LIN {X 151.987,Y 68.741,Z 52.000,A 180.000,B 0.000,C 180.000} C_DIS
LIN {X 152.500,Y 68.741,Z 52.000,A 180.000,B 0.000,C 180.000} C_DIS
LIN {X 152.500,Y 68.741,Z 45.000,A 180.000,B 0.000,C 180.000} C_DIS
LIN {X 155.010,Y 68.741,Z 45.000,A 180.000,B 0.000,C 180.000} C_DIS
; Link Move Starts
LIN {X 155.120,Y 68.741,Z 45.026,A 180.000,B 0.000,C 180.000} C_DIS
LIN {X 155.230,Y 68.741,Z 45.051,A 180.000,B 0.000,C 180.000} C_DIS
LIN {X 155.771,Y 69.054,Z 45.051,A 180.000,B 0.000,C 180.000} C_DIS
LIN {X 155.771,Y 69.679,Z 45.051,A 180.000,B 0.000,C 180.000} C_DIS
LIN {X 155.230,Y 69.991,Z 45.051,A 180.000,B 0.000,C 180.000} C_DIS
LIN {X 155.120,Y 69.991,Z 45.026,A 180.000,B 0.000,C 180.000} C_DIS
LIN {X 155.010,Y 69.991,Z 45.000,A 180.000,B 0.000,C 180.000} C_DIS
; Cutting Move Starts
LIN {X 152.500,Y 69.991,Z 45.000,A 180.000,B 0.000,C 180.000} C_DIS
LIN {X 152.500,Y 69.991,Z 52.000,A 180.000,B 0.000,C 180.000} C_DIS
LIN {X 152.119,Y 69.991,Z 52.000,A 180.000,B 0.000,C 180.000} C_DIS
LIN {X 152.117,Y 69.991,Z 57.000,A 180.000,B 0.000,C 180.000} C_DIS
LIN {X 138.527,Y 69.991,Z 57.000,A 180.000,B 0.000,C 180.000} C_DIS
LIN {X 138.527,Y 69.991,Z 62.000,A 180.000,B 0.000,C 180.000} C_DIS
LIN {X 64.935,Y 69.991,Z 62.000,A 180.000,B 0.000,C 180.000} C_DIS
LIN {X 64.931,Y 69.991,Z 82.040,A 180.000,B 0.000,C 180.000} C_DIS
LIN {X 64.891,Y 69.991,Z 82.144,A 180.000,B 0.000,C 180.000} C_DIS
LIN {X 64.812,Y 69.991,Z 82.250,A 180.000,B 0.000,C 180.000} C_DIS
LIN {X 64.651,Y 69.991,Z 82.406,A 180.000,B 0.000,C 180.000} C_DIS
LIN {X 64.413,Y 69.991,Z 82.569,A 180.000,B 0.000,C 180.000} C_DIS
LIN {X 64.256,Y 69.991,Z 82.658,A 180.000,B 0.000,C 180.000} C_DIS
LIN {X 63.886,Y 69.991,Z 82.826,A 180.000,B 0.000,C 180.000} C_DIS
LIN {X 63.427,Y 69.991,Z 82.974,A 180.000,B 0.000,C 180.000} C_DIS
LIN {X 63.116,Y 69.991,Z 83.044,A 180.000,B 0.000,C 180.000} C_DIS
LIN {X 62.751,Y 69.991,Z 83.103,A 180.000,B 0.000,C 180.000} C_DIS
LIN {X 62.375,Y 69.991,Z 83.137,A 180.000,B 0.000,C 180.000} C_DIS
LIN {X 62.046,Y 69.991,Z 83.148,A 180.000,B 0.000,C 180.000} C_DIS
LIN {X 57.054,Y 69.991,Z 83.146,A 180.000,B 0.000,C 180.000} C_DIS
LIN {X 56.742,Y 69.991,Z 83.135,A 180.000,B 0.000,C 180.000} C_DIS
LIN {X 56.417,Y 69.991,Z 83.115,A 180.000,B 0.000,C 180.000} C_DIS
LIN {X 56.096,Y 69.991,Z 83.085,A 180.000,B 0.000,C 180.000} C_DIS
LIN {X 55.739,Y 69.991,Z 83.040,A 180.000,B 0.000,C 180.000} C_DIS
LIN {X 55.361,Y 69.991,Z 82.981,A 180.000,B 0.000,C 180.000} C_DIS
LIN {X 55.002,Y 69.991,Z 82.912,A 180.000,B 0.000,C 180.000} C_DIS
LIN {X 54.625,Y 69.991,Z 82.827,A 180.000,B 0.000,C 180.000} C_DIS
LIN {X 54.239,Y 69.991,Z 82.728,A 180.000,B 0.000,C 180.000} C_DIS
LIN {X 53.862,Y 69.991,Z 82.617,A 180.000,B 0.000,C 180.000} C_DIS
LIN {X 53.473,Y 69.991,Z 82.491,A 180.000,B 0.000,C 180.000} C_DIS
LIN {X 53.083,Y 69.991,Z 82.351,A 180.000,B 0.000,C 180.000} C_DIS
LIN {X 52.690,Y 69.991,Z 82.196,A 180.000,B 0.000,C 180.000} C_DIS
LIN {X 52.293,Y 69.991,Z 82.027,A 180.000,B 0.000,C 180.000} C_DIS
LIN {X 51.893,Y 69.991,Z 81.843,A 180.000,B 0.000,C 180.000} C_DIS
LIN {X 51.488,Y 69.991,Z 81.643,A 180.000,B 0.000,C 180.000} C_DIS
LIN {X 51.080,Y 69.991,Z 81.428,A 180.000,B 0.000,C 180.000} C_DIS
LIN {X 50.671,Y 69.991,Z 81.199,A 180.000,B 0.000,C 180.000} C_DIS
LIN {X 50.251,Y 69.991,Z 80.950,A 180.000,B 0.000,C 180.000} C_DIS
LIN {X 49.826,Y 69.991,Z 80.683,A 180.000,B 0.000,C 180.000} C_DIS
LIN {X 49.494,Y 69.991,Z 80.467,A 180.000,B 0.000,C 180.000} C_DIS
LIN {X 49.494,Y 69.991,Z 62.000,A 180.000,B 0.000,C 180.000} C_DIS
LIN {X 16.473,Y 69.991,Z 62.000,A 180.000,B 0.000,C 180.000} C_DIS
LIN {X 16.473,Y 69.991,Z 57.000,A 180.000,B 0.000,C 180.000} C_DIS
LIN {X 2.881,Y 69.991,Z 57.000,A 180.000,B 0.000,C 180.000} C_DIS
LIN {X 2.881,Y 69.991,Z 52.000,A 180.000,B 0.000,C 180.000} C_DIS
LIN {X 2.500,Y 69.991,Z 52.000,A 180.000,B 0.000,C 180.000} C_DIS
LIN {X 2.500,Y 69.991,Z 45.000,A 180.000,B 0.000,C 180.000} C_DIS
LIN {X -0.010,Y 69.991,Z 45.000,A 180.000,B 0.000,C 180.000} C_DIS
; Link Move Starts
LIN {X -0.120,Y 69.991,Z 45.026,A 180.000,B 0.000,C 180.000} C_DIS
LIN {X -0.230,Y 69.991,Z 45.051,A 180.000,B 0.000,C 180.000} C_DIS
LIN {X -0.771,Y 70.304,Z 45.051,A 180.000,B 0.000,C 180.000} C_DIS
LIN {X -0.771,Y 70.929,Z 45.051,A 180.000,B 0.000,C 180.000} C_DIS
LIN {X -0.230,Y 71.241,Z 45.051,A 180.000,B 0.000,C 180.000} C_DIS
LIN {X -0.120,Y 71.241,Z 45.026,A 180.000,B 0.000,C 180.000} C_DIS
LIN {X -0.010,Y 71.241,Z 45.000,A 180.000,B 0.000,C 180.000} C_DIS
; Cutting Move Starts
LIN {X 2.500,Y 71.241,Z 45.000,A 180.000,B 0.000,C 180.000} C_DIS
LIN {X 2.500,Y 71.241,Z 52.000,A 180.000,B 0.000,C 180.000} C_DIS
LIN {X 2.765,Y 71.241,Z 52.000,A 180.000,B 0.000,C 180.000} C_DIS
LIN {X 2.767,Y 71.241,Z 57.000,A 180.000,B 0.000,C 180.000} C_DIS
LIN {X 15.220,Y 71.241,Z 57.000,A 180.000,B 0.000,C 180.000} C_DIS
LIN {X 15.224,Y 71.241,Z 62.000,A 180.000,B 0.000,C 180.000} C_DIS
LIN {X 49.913,Y 71.241,Z 62.000,A 180.000,B 0.000,C 180.000} C_DIS
LIN {X 49.916,Y 71.241,Z 80.467,A 180.000,B 0.000,C 180.000} C_DIS
LIN {X 50.252,Y 71.241,Z 80.686,A 180.000,B 0.000,C 180.000} C_DIS
LIN {X 50.672,Y 71.241,Z 80.949,A 180.000,B 0.000,C 180.000} C_DIS
LIN {X 51.086,Y 71.241,Z 81.195,A 180.000,B 0.000,C 180.000} C_DIS
LIN {X 51.500,Y 71.241,Z 81.427,A 180.000,B 0.000,C 180.000} C_DIS
LIN {X 51.909,Y 71.241,Z 81.643,A 180.000,B 0.000,C 180.000} C_DIS
LIN {X 52.314,Y 71.241,Z 81.842,A 180.000,B 0.000,C 180.000} C_DIS
LIN {X 52.714,Y 71.241,Z 82.026,A 180.000,B 0.000,C 180.000} C_DIS
LIN {X 53.057,Y 71.241,Z 82.173,A 180.000,B 0.000,C 180.000} C_DIS
LIN {X 53.316,Y 71.241,Z 82.278,A 180.000,B 0.000,C 180.000} C_DIS
LIN {X 53.758,Y 71.241,Z 82.442,A 180.000,B 0.000,C 180.000} C_DIS
LIN {X 54.177,Y 71.241,Z 82.579,A 180.000,B 0.000,C 180.000} C_DIS
LIN {X 54.617,Y 71.241,Z 82.706,A 180.000,B 0.000,C 180.000} C_DIS
LIN {X 55.075,Y 71.241,Z 82.819,A 180.000,B 0.000,C 180.000} C_DIS
LIN {X 55.690,Y 71.241,Z 82.942,A 180.000,B 0.000,C 180.000} C_DIS
LIN {X 56.199,Y 71.241,Z 83.020,A 180.000,B 0.000,C 180.000} C_DIS
LIN {X 56.683,Y 71.241,Z 83.076,A 180.000,B 0.000,C 180.000} C_DIS
LIN {X 57.277,Y 71.241,Z 83.123,A 180.000,B 0.000,C 180.000} C_DIS
LIN {X 57.978,Y 71.241,Z 83.146,A 180.000,B 0.000,C 180.000} C_DIS
LIN {X 61.059,Y 71.241,Z 83.147,A 180.000,B 0.000,C 180.000} C_DIS
LIN {X 61.178,Y 71.241,Z 83.135,A 180.000,B 0.000,C 180.000} C_DIS
LIN {X 61.226,Y 71.241,Z 83.119,A 180.000,B 0.000,C 180.000} C_DIS
LIN {X 61.230,Y 71.241,Z 62.000,A 180.000,B 0.000,C 180.000} C_DIS
LIN {X 73.375,Y 71.241,Z 62.000,A 180.000,B 0.000,C 180.000} C_DIS
LIN {X 73.375,Y 71.241,Z 57.000,A 180.000,B 0.000,C 180.000} C_DIS
LIN {X 81.625,Y 71.241,Z 57.000,A 180.000,B 0.000,C 180.000} C_DIS
LIN {X 81.625,Y 71.241,Z 62.000,A 180.000,B 0.000,C 180.000} C_DIS
LIN {X 139.775,Y 71.241,Z 62.000,A 180.000,B 0.000,C 180.000} C_DIS
LIN {X 139.777,Y 71.241,Z 57.000,A 180.000,B 0.000,C 180.000} C_DIS
LIN {X 152.233,Y 71.241,Z 57.000,A 180.000,B 0.000,C 180.000} C_DIS
LIN {X 152.233,Y 71.241,Z 52.000,A 180.000,B 0.000,C 180.000} C_DIS
LIN {X 152.500,Y 71.241,Z 52.000,A 180.000,B 0.000,C 180.000} C_DIS
LIN {X 152.500,Y 71.241,Z 45.000,A 180.000,B 0.000,C 180.000} C_DIS
LIN {X 155.010,Y 71.241,Z 45.000,A 180.000,B 0.000,C 180.000} C_DIS
; Link Move Starts
LIN {X 155.120,Y 71.241,Z 45.026,A 180.000,B 0.000,C 180.000} C_DIS
LIN {X 155.230,Y 71.241,Z 45.051,A 180.000,B 0.000,C 180.000} C_DIS
LIN {X 155.771,Y 71.553,Z 45.051,A 180.000,B 0.000,C 180.000} C_DIS
LIN {X 155.771,Y 72.178,Z 45.051,A 180.000,B 0.000,C 180.000} C_DIS
LIN {X 155.230,Y 72.491,Z 45.051,A 180.000,B 0.000,C 180.000} C_DIS
LIN {X 155.120,Y 72.491,Z 45.026,A 180.000,B 0.000,C 180.000} C_DIS
LIN {X 155.010,Y 72.491,Z 45.000,A 180.000,B 0.000,C 180.000} C_DIS
; Cutting Move Starts
LIN {X 152.500,Y 72.491,Z 45.000,A 180.000,B 0.000,C 180.000} C_DIS
LIN {X 152.500,Y 72.491,Z 52.000,A 180.000,B 0.000,C 180.000} C_DIS
LIN {X 152.330,Y 72.491,Z 52.000,A 180.000,B 0.000,C 180.000} C_DIS
LIN {X 152.330,Y 72.491,Z 57.000,A 180.000,B 0.000,C 180.000} C_DIS
LIN {X 141.026,Y 72.491,Z 57.000,A 180.000,B 0.000,C 180.000} C_DIS
LIN {X 141.026,Y 72.491,Z 62.000,A 180.000,B 0.000,C 180.000} C_DIS
LIN {X 83.076,Y 72.491,Z 62.000,A 180.000,B 0.000,C 180.000} C_DIS
LIN {X 83.076,Y 72.491,Z 57.000,A 180.000,B 0.000,C 180.000} C_DIS
LIN {X 71.924,Y 72.491,Z 57.000,A 180.000,B 0.000,C 180.000} C_DIS
LIN {X 71.924,Y 72.491,Z 62.000,A 180.000,B 0.000,C 180.000} C_DIS
LIN {X 57.525,Y 72.491,Z 62.000,A 180.000,B 0.000,C 180.000} C_DIS
LIN {X 57.521,Y 72.491,Z 82.696,A 180.000,B 0.000,C 180.000} C_DIS
LIN {X 57.489,Y 72.491,Z 82.734,A 180.000,B 0.000,C 180.000} C_DIS
LIN {X 57.421,Y 72.491,Z 82.763,A 180.000,B 0.000,C 180.000} C_DIS
LIN {X 57.262,Y 72.491,Z 82.785,A 180.000,B 0.000,C 180.000} C_DIS
LIN {X 56.970,Y 72.491,Z 82.787,A 180.000,B 0.000,C 180.000} C_DIS
LIN {X 56.506,Y 72.491,Z 82.752,A 180.000,B 0.000,C 180.000} C_DIS
LIN {X 55.884,Y 72.491,Z 82.665,A 180.000,B 0.000,C 180.000} C_DIS
LIN {X 55.297,Y 72.491,Z 82.553,A 180.000,B 0.000,C 180.000} C_DIS
LIN {X 54.770,Y 72.491,Z 82.429,A 180.000,B 0.000,C 180.000} C_DIS
LIN {X 54.285,Y 72.491,Z 82.296,A 180.000,B 0.000,C 180.000} C_DIS
LIN {X 53.823,Y 72.491,Z 82.152,A 180.000,B 0.000,C 180.000} C_DIS
LIN {X 53.356,Y 72.491,Z 81.988,A 180.000,B 0.000,C 180.000} C_DIS
LIN {X 52.884,Y 72.491,Z 81.804,A 180.000,B 0.000,C 180.000} C_DIS
LIN {X 52.420,Y 72.491,Z 81.604,A 180.000,B 0.000,C 180.000} C_DIS
LIN {X 51.957,Y 72.491,Z 81.385,A 180.000,B 0.000,C 180.000} C_DIS
LIN {X 51.493,Y 72.491,Z 81.145,A 180.000,B 0.000,C 180.000} C_DIS
LIN {X 51.033,Y 72.491,Z 80.888,A 180.000,B 0.000,C 180.000} C_DIS
LIN {X 50.578,Y 72.491,Z 80.613,A 180.000,B 0.000,C 180.000} C_DIS
LIN {X 50.346,Y 72.491,Z 80.467,A 180.000,B 0.000,C 180.000} C_DIS
LIN {X 50.346,Y 72.491,Z 62.000,A 180.000,B 0.000,C 180.000} C_DIS
LIN {X 13.974,Y 72.491,Z 62.000,A 180.000,B 0.000,C 180.000} C_DIS
LIN {X 13.974,Y 72.491,Z 57.000,A 180.000,B 0.000,C 180.000} C_DIS
LIN {X 2.670,Y 72.491,Z 57.000,A 180.000,B 0.000,C 180.000} C_DIS
LIN {X 2.670,Y 72.491,Z 52.000,A 180.000,B 0.000,C 180.000} C_DIS
LIN {X 2.500,Y 72.491,Z 52.000,A 180.000,B 0.000,C 180.000} C_DIS
LIN {X 2.495,Y 72.491,Z 45.000,A 180.000,B 0.000,C 180.000} C_DIS
LIN {X -0.010,Y 72.491,Z 45.000,A 180.000,B 0.000,C 180.000} C_DIS
; Link Move Starts
LIN {X -0.120,Y 72.491,Z 45.026,A 180.000,B 0.000,C 180.000} C_DIS
LIN {X -0.230,Y 72.491,Z 45.051,A 180.000,B 0.000,C 180.000} C_DIS
LIN {X -0.771,Y 72.803,Z 45.051,A 180.000,B 0.000,C 180.000} C_DIS
LIN {X -0.771,Y 73.428,Z 45.051,A 180.000,B 0.000,C 180.000} C_DIS
LIN {X -0.230,Y 73.741,Z 45.051,A 180.000,B 0.000,C 180.000} C_DIS
LIN {X -0.120,Y 73.741,Z 45.026,A 180.000,B 0.000,C 180.000} C_DIS
LIN {X -0.010,Y 73.741,Z 45.000,A 180.000,B 0.000,C 180.000} C_DIS
; Cutting Move Starts
LIN {X 2.500,Y 73.741,Z 45.000,A 180.000,B 0.000,C 180.000} C_DIS
LIN {X 2.500,Y 73.741,Z 52.000,A 180.000,B 0.000,C 180.000} C_DIS
LIN {X 2.597,Y 73.741,Z 52.000,A 180.000,B 0.000,C 180.000} C_DIS
LIN {X 2.597,Y 73.741,Z 57.000,A 180.000,B 0.000,C 180.000} C_DIS
LIN {X 12.724,Y 73.741,Z 57.000,A 180.000,B 0.000,C 180.000} C_DIS
LIN {X 12.724,Y 73.741,Z 62.000,A 180.000,B 0.000,C 180.000} C_DIS
LIN {X 51.532,Y 73.741,Z 62.000,A 180.000,B 0.000,C 180.000} C_DIS
LIN {X 51.533,Y 73.741,Z 80.467,A 180.000,B 0.000,C 180.000} C_DIS
LIN {X 51.861,Y 73.741,Z 80.604,A 180.000,B 0.000,C 180.000} C_DIS
LIN {X 52.317,Y 73.741,Z 80.775,A 180.000,B 0.000,C 180.000} C_DIS
LIN {X 52.750,Y 73.741,Z 80.905,A 180.000,B 0.000,C 180.000} C_DIS
LIN {X 53.082,Y 73.741,Z 80.979,A 180.000,B 0.000,C 180.000} C_DIS
LIN {X 53.328,Y 73.741,Z 81.008,A 180.000,B 0.000,C 180.000} C_DIS
LIN {X 53.527,Y 73.741,Z 81.004,A 180.000,B 0.000,C 180.000} C_DIS
LIN {X 53.649,Y 73.741,Z 80.977,A 180.000,B 0.000,C 180.000} C_DIS
LIN {X 53.735,Y 73.741,Z 80.931,A 180.000,B 0.000,C 180.000} C_DIS
LIN {X 53.786,Y 73.741,Z 80.873,A 180.000,B 0.000,C 180.000} C_DIS
LIN {X 53.816,Y 73.741,Z 80.795,A 180.000,B 0.000,C 180.000} C_DIS
LIN {X 53.820,Y 73.741,Z 62.000,A 180.000,B 0.000,C 180.000} C_DIS
LIN {X 71.016,Y 73.741,Z 62.000,A 180.000,B 0.000,C 180.000} C_DIS
LIN {X 71.016,Y 73.741,Z 57.000,A 180.000,B 0.000,C 180.000} C_DIS
LIN {X 83.984,Y 73.741,Z 57.000,A 180.000,B 0.000,C 180.000} C_DIS
LIN {X 83.984,Y 73.741,Z 62.000,A 180.000,B 0.000,C 180.000} C_DIS
LIN {X 142.272,Y 73.741,Z 62.000,A 180.000,B 0.000,C 180.000} C_DIS
LIN {X 142.276,Y 73.741,Z 57.000,A 180.000,B 0.000,C 180.000} C_DIS
LIN {X 152.403,Y 73.741,Z 57.000,A 180.000,B 0.000,C 180.000} C_DIS
LIN {X 152.403,Y 73.741,Z 52.000,A 180.000,B 0.000,C 180.000} C_DIS
LIN {X 152.500,Y 73.741,Z 52.000,A 180.000,B 0.000,C 180.000} C_DIS
LIN {X 152.500,Y 73.741,Z 45.000,A 180.000,B 0.000,C 180.000} C_DIS
LIN {X 155.010,Y 73.741,Z 45.000,A 180.000,B 0.000,C 180.000} C_DIS
; Link Move Starts
LIN {X 155.120,Y 73.741,Z 45.026,A 180.000,B 0.000,C 180.000} C_DIS
LIN {X 155.230,Y 73.741,Z 45.051,A 180.000,B 0.000,C 180.000} C_DIS
LIN {X 155.771,Y 74.053,Z 45.051,A 180.000,B 0.000,C 180.000} C_DIS
LIN {X 155.771,Y 74.678,Z 45.051,A 180.000,B 0.000,C 180.000} C_DIS
LIN {X 155.230,Y 74.991,Z 45.051,A 180.000,B 0.000,C 180.000} C_DIS
LIN {X 155.120,Y 74.991,Z 45.026,A 180.000,B 0.000,C 180.000} C_DIS
LIN {X 155.010,Y 74.991,Z 45.000,A 180.000,B 0.000,C 180.000} C_DIS
; Cutting Move Starts
LIN {X 152.500,Y 74.991,Z 45.000,A 180.000,B 0.000,C 180.000} C_DIS
LIN {X 152.500,Y 74.991,Z 52.000,A 180.000,B 0.000,C 180.000} C_DIS
LIN {X 152.453,Y 74.991,Z 52.000,A 180.000,B 0.000,C 180.000} C_DIS
LIN {X 152.453,Y 74.991,Z 57.000,A 180.000,B 0.000,C 180.000} C_DIS
LIN {X 143.526,Y 74.991,Z 57.000,A 180.000,B 0.000,C 180.000} C_DIS
LIN {X 143.526,Y 74.991,Z 62.000,A 180.000,B 0.000,C 180.000} C_DIS
LIN {X 84.563,Y 74.991,Z 62.000,A 180.000,B 0.000,C 180.000} C_DIS
LIN {X 84.563,Y 74.991,Z 57.000,A 180.000,B 0.000,C 180.000} C_DIS
LIN {X 70.437,Y 74.991,Z 57.000,A 180.000,B 0.000,C 180.000} C_DIS
LIN {X 70.436,Y 74.991,Z 62.000,A 180.000,B 0.000,C 180.000} C_DIS
LIN {X 11.474,Y 74.991,Z 62.000,A 180.000,B 0.000,C 180.000} C_DIS
LIN {X 11.474,Y 74.991,Z 57.000,A 180.000,B 0.000,C 180.000} C_DIS
LIN {X 2.547,Y 74.991,Z 57.000,A 180.000,B 0.000,C 180.000} C_DIS
LIN {X 2.547,Y 74.991,Z 52.000,A 180.000,B 0.000,C 180.000} C_DIS
LIN {X 2.500,Y 74.991,Z 52.000,A 180.000,B 0.000,C 180.000} C_DIS
LIN {X 2.500,Y 74.991,Z 45.000,A 180.000,B 0.000,C 180.000} C_DIS
LIN {X -0.010,Y 74.991,Z 45.000,A 180.000,B 0.000,C 180.000} C_DIS
; Link Move Starts
LIN {X -0.120,Y 74.991,Z 45.026,A 180.000,B 0.000,C 180.000} C_DIS
LIN {X -0.230,Y 74.991,Z 45.051,A 180.000,B 0.000,C 180.000} C_DIS
LIN {X -0.771,Y 75.303,Z 45.051,A 180.000,B 0.000,C 180.000} C_DIS
LIN {X -0.771,Y 75.928,Z 45.051,A 180.000,B 0.000,C 180.000} C_DIS
LIN {X -0.230,Y 76.241,Z 45.051,A 180.000,B 0.000,C 180.000} C_DIS
LIN {X -0.120,Y 76.241,Z 45.026,A 180.000,B 0.000,C 180.000} C_DIS
LIN {X -0.010,Y 76.241,Z 45.000,A 180.000,B 0.000,C 180.000} C_DIS
; Cutting Move Starts
LIN {X 2.500,Y 76.241,Z 45.000,A 180.000,B 0.000,C 180.000} C_DIS
LIN {X 2.500,Y 76.241,Z 52.000,A 180.000,B 0.000,C 180.000} C_DIS
LIN {X 2.515,Y 76.241,Z 52.000,A 180.000,B 0.000,C 180.000} C_DIS
LIN {X 2.515,Y 76.241,Z 57.000,A 180.000,B 0.000,C 180.000} C_DIS
LIN {X 10.340,Y 76.241,Z 57.000,A 180.000,B 0.000,C 180.000} C_DIS
LIN {X 10.340,Y 76.241,Z 62.000,A 180.000,B 0.000,C 180.000} C_DIS
LIN {X 70.111,Y 76.241,Z 62.000,A 180.000,B 0.000,C 180.000} C_DIS
LIN {X 70.111,Y 76.241,Z 57.000,A 180.000,B 0.000,C 180.000} C_DIS
LIN {X 84.889,Y 76.241,Z 57.000,A 180.000,B 0.000,C 180.000} C_DIS
LIN {X 84.889,Y 76.241,Z 62.000,A 180.000,B 0.000,C 180.000} C_DIS
LIN {X 144.660,Y 76.241,Z 62.000,A 180.000,B 0.000,C 180.000} C_DIS
LIN {X 144.660,Y 76.241,Z 57.000,A 180.000,B 0.000,C 180.000} C_DIS
LIN {X 152.484,Y 76.241,Z 57.000,A 180.000,B 0.000,C 180.000} C_DIS
LIN {X 152.485,Y 76.241,Z 52.000,A 180.000,B 0.000,C 180.000} C_DIS
LIN {X 152.500,Y 76.241,Z 52.000,A 180.000,B 0.000,C 180.000} C_DIS
LIN {X 152.500,Y 76.241,Z 45.000,A 180.000,B 0.000,C 180.000} C_DIS
LIN {X 155.010,Y 76.241,Z 45.000,A 180.000,B 0.000,C 180.000} C_DIS
; Link Move Starts
LIN {X 155.120,Y 76.241,Z 45.026,A 180.000,B 0.000,C 180.000} C_DIS
LIN {X 155.230,Y 76.241,Z 45.051,A 180.000,B 0.000,C 180.000} C_DIS
LIN {X 155.771,Y 76.553,Z 45.051,A 180.000,B 0.000,C 180.000} C_DIS
LIN {X 155.771,Y 77.178,Z 45.051,A 180.000,B 0.000,C 180.000} C_DIS
LIN {X 155.230,Y 77.490,Z 45.051,A 180.000,B 0.000,C 180.000} C_DIS
LIN {X 155.120,Y 77.490,Z 45.026,A 180.000,B 0.000,C 180.000} C_DIS
LIN {X 155.010,Y 77.490,Z 45.000,A 180.000,B 0.000,C 180.000} C_DIS
; Cutting Move Starts
LIN {X 152.500,Y 77.490,Z 45.000,A 180.000,B 0.000,C 180.000} C_DIS
LIN {X 152.500,Y 77.490,Z 57.000,A 180.000,B 0.000,C 180.000} C_DIS
LIN {X 145.000,Y 77.490,Z 57.000,A 180.000,B 0.000,C 180.000} C_DIS
LIN {X 145.000,Y 77.490,Z 62.000,A 180.000,B 0.000,C 180.000} C_DIS
LIN {X 84.998,Y 77.490,Z 62.000,A 180.000,B 0.000,C 180.000} C_DIS
LIN {X 84.998,Y 77.490,Z 57.000,A 180.000,B 0.000,C 180.000} C_DIS
LIN {X 70.002,Y 77.490,Z 57.000,A 180.000,B 0.000,C 180.000} C_DIS
LIN {X 70.000,Y 77.490,Z 62.000,A 180.000,B 0.000,C 180.000} C_DIS
LIN {X 10.000,Y 77.490,Z 62.000,A 180.000,B 0.000,C 180.000} C_DIS
LIN {X 10.000,Y 77.490,Z 57.000,A 180.000,B 0.000,C 180.000} C_DIS
LIN {X 2.500,Y 77.490,Z 57.000,A 180.000,B 0.000,C 180.000} C_DIS
LIN {X 2.500,Y 77.490,Z 45.000,A 180.000,B 0.000,C 180.000} C_DIS
LIN {X -0.010,Y 77.490,Z 45.000,A 180.000,B 0.000,C 180.000} C_DIS
; Link Move Starts
LIN {X -0.120,Y 77.490,Z 45.026,A 180.000,B 0.000,C 180.000} C_DIS
LIN {X -0.230,Y 77.490,Z 45.051,A 180.000,B 0.000,C 180.000} C_DIS
LIN {X -0.771,Y 77.803,Z 45.051,A 180.000,B 0.000,C 180.000} C_DIS
LIN {X -0.771,Y 78.428,Z 45.051,A 180.000,B 0.000,C 180.000} C_DIS
LIN {X -0.230,Y 78.740,Z 45.051,A 180.000,B 0.000,C 180.000} C_DIS
LIN {X -0.120,Y 78.740,Z 45.026,A 180.000,B 0.000,C 180.000} C_DIS
LIN {X -0.010,Y 78.740,Z 45.000,A 180.000,B 0.000,C 180.000} C_DIS
; Cutting Move Starts
LIN {X 2.500,Y 78.740,Z 45.000,A 180.000,B 0.000,C 180.000} C_DIS
LIN {X 2.500,Y 78.740,Z 52.000,A 180.000,B 0.000,C 180.000} C_DIS
LIN {X 2.514,Y 78.740,Z 52.000,A 180.000,B 0.000,C 180.000} C_DIS
LIN {X 2.514,Y 78.740,Z 57.000,A 180.000,B 0.000,C 180.000} C_DIS
LIN {X 10.328,Y 78.740,Z 57.000,A 180.000,B 0.000,C 180.000} C_DIS
LIN {X 10.329,Y 78.740,Z 62.000,A 180.000,B 0.000,C 180.000} C_DIS
LIN {X 70.108,Y 78.740,Z 62.000,A 180.000,B 0.000,C 180.000} C_DIS
LIN {X 70.108,Y 78.740,Z 57.000,A 180.000,B 0.000,C 180.000} C_DIS
LIN {X 84.890,Y 78.740,Z 57.000,A 180.000,B 0.000,C 180.000} C_DIS
LIN {X 84.892,Y 78.740,Z 62.000,A 180.000,B 0.000,C 180.000} C_DIS
LIN {X 144.671,Y 78.740,Z 62.000,A 180.000,B 0.000,C 180.000} C_DIS
LIN {X 144.671,Y 78.740,Z 57.000,A 180.000,B 0.000,C 180.000} C_DIS
LIN {X 152.484,Y 78.740,Z 57.000,A 180.000,B 0.000,C 180.000} C_DIS
LIN {X 152.486,Y 78.740,Z 52.000,A 180.000,B 0.000,C 180.000} C_DIS
LIN {X 152.500,Y 78.740,Z 52.000,A 180.000,B 0.000,C 180.000} C_DIS
LIN {X 152.500,Y 78.740,Z 45.000,A 180.000,B 0.000,C 180.000} C_DIS
LIN {X 155.010,Y 78.740,Z 45.000,A 180.000,B 0.000,C 180.000} C_DIS
; Link Move Starts
LIN {X 155.120,Y 78.740,Z 45.026,A 180.000,B 0.000,C 180.000} C_DIS
LIN {X 155.230,Y 78.740,Z 45.051,A 180.000,B 0.000,C 180.000} C_DIS
LIN {X 155.771,Y 79.053,Z 45.051,A 180.000,B 0.000,C 180.000} C_DIS
LIN {X 155.771,Y 79.678,Z 45.051,A 180.000,B 0.000,C 180.000} C_DIS
LIN {X 155.230,Y 79.990,Z 45.051,A 180.000,B 0.000,C 180.000} C_DIS
LIN {X 155.120,Y 79.990,Z 45.026,A 180.000,B 0.000,C 180.000} C_DIS
LIN {X 155.010,Y 79.990,Z 45.000,A 180.000,B 0.000,C 180.000} C_DIS
; Cutting Move Starts
LIN {X 152.500,Y 79.990,Z 45.000,A 180.000,B 0.000,C 180.000} C_DIS
LIN {X 152.500,Y 79.990,Z 52.000,A 180.000,B 0.000,C 180.000} C_DIS
LIN {X 152.454,Y 79.990,Z 52.000,A 180.000,B 0.000,C 180.000} C_DIS
LIN {X 152.454,Y 79.990,Z 57.000,A 180.000,B 0.000,C 180.000} C_DIS
LIN {X 143.545,Y 79.990,Z 57.000,A 180.000,B 0.000,C 180.000} C_DIS
LIN {X 143.545,Y 79.990,Z 62.000,A 180.000,B 0.000,C 180.000} C_DIS
LIN {X 84.569,Y 79.990,Z 62.000,A 180.000,B 0.000,C 180.000} C_DIS
LIN {X 84.569,Y 79.990,Z 57.000,A 180.000,B 0.000,C 180.000} C_DIS
LIN {X 70.431,Y 79.990,Z 57.000,A 180.000,B 0.000,C 180.000} C_DIS
LIN {X 70.428,Y 79.990,Z 62.000,A 180.000,B 0.000,C 180.000} C_DIS
LIN {X 11.455,Y 79.990,Z 62.000,A 180.000,B 0.000,C 180.000} C_DIS
LIN {X 11.455,Y 79.990,Z 57.000,A 180.000,B 0.000,C 180.000} C_DIS
LIN {X 2.546,Y 79.990,Z 57.000,A 180.000,B 0.000,C 180.000} C_DIS
LIN {X 2.546,Y 79.990,Z 52.000,A 180.000,B 0.000,C 180.000} C_DIS
LIN {X 2.500,Y 79.990,Z 52.000,A 180.000,B 0.000,C 180.000} C_DIS
LIN {X 2.500,Y 79.990,Z 45.000,A 180.000,B 0.000,C 180.000} C_DIS
LIN {X -0.010,Y 79.990,Z 45.000,A 180.000,B 0.000,C 180.000} C_DIS
; Link Move Starts
LIN {X -0.120,Y 79.990,Z 45.026,A 180.000,B 0.000,C 180.000} C_DIS
LIN {X -0.230,Y 79.990,Z 45.051,A 180.000,B 0.000,C 180.000} C_DIS
LIN {X -0.771,Y 80.303,Z 45.051,A 180.000,B 0.000,C 180.000} C_DIS
LIN {X -0.771,Y 80.928,Z 45.051,A 180.000,B 0.000,C 180.000} C_DIS
LIN {X -0.230,Y 81.240,Z 45.051,A 180.000,B 0.000,C 180.000} C_DIS
LIN {X -0.120,Y 81.240,Z 45.026,A 180.000,B 0.000,C 180.000} C_DIS
LIN {X -0.010,Y 81.240,Z 45.000,A 180.000,B 0.000,C 180.000} C_DIS
; Cutting Move Starts
LIN {X 2.500,Y 81.240,Z 45.000,A 180.000,B 0.000,C 180.000} C_DIS
LIN {X 2.500,Y 81.240,Z 52.000,A 180.000,B 0.000,C 180.000} C_DIS
LIN {X 2.595,Y 81.240,Z 52.000,A 180.000,B 0.000,C 180.000} C_DIS
LIN {X 2.595,Y 81.240,Z 57.000,A 180.000,B 0.000,C 180.000} C_DIS
LIN {X 12.705,Y 81.240,Z 57.000,A 180.000,B 0.000,C 180.000} C_DIS
LIN {X 12.705,Y 81.240,Z 62.000,A 180.000,B 0.000,C 180.000} C_DIS
LIN {X 71.002,Y 81.240,Z 62.000,A 180.000,B 0.000,C 180.000} C_DIS
LIN {X 71.004,Y 81.240,Z 57.000,A 180.000,B 0.000,C 180.000} C_DIS
LIN {X 83.996,Y 81.240,Z 57.000,A 180.000,B 0.000,C 180.000} C_DIS
LIN {X 83.996,Y 81.240,Z 62.000,A 180.000,B 0.000,C 180.000} C_DIS
LIN {X 142.295,Y 81.240,Z 62.000,A 180.000,B 0.000,C 180.000} C_DIS
LIN {X 142.295,Y 81.240,Z 57.000,A 180.000,B 0.000,C 180.000} C_DIS
LIN {X 152.405,Y 81.240,Z 57.000,A 180.000,B 0.000,C 180.000} C_DIS
LIN {X 152.405,Y 81.240,Z 52.000,A 180.000,B 0.000,C 180.000} C_DIS
LIN {X 152.500,Y 81.240,Z 52.000,A 180.000,B 0.000,C 180.000} C_DIS
LIN {X 152.500,Y 81.240,Z 45.000,A 180.000,B 0.000,C 180.000} C_DIS
LIN {X 155.010,Y 81.240,Z 45.000,A 180.000,B 0.000,C 180.000} C_DIS
; Link Move Starts
LIN {X 155.120,Y 81.240,Z 45.026,A 180.000,B 0.000,C 180.000} C_DIS
LIN {X 155.230,Y 81.240,Z 45.051,A 180.000,B 0.000,C 180.000} C_DIS
LIN {X 155.771,Y 81.553,Z 45.051,A 180.000,B 0.000,C 180.000} C_DIS
LIN {X 155.771,Y 82.178,Z 45.051,A 180.000,B 0.000,C 180.000} C_DIS
LIN {X 155.230,Y 82.490,Z 45.051,A 180.000,B 0.000,C 180.000} C_DIS
LIN {X 155.120,Y 82.490,Z 45.026,A 180.000,B 0.000,C 180.000} C_DIS
LIN {X 155.010,Y 82.490,Z 45.000,A 180.000,B 0.000,C 180.000} C_DIS
; Cutting Move Starts
LIN {X 152.500,Y 82.490,Z 45.000,A 180.000,B 0.000,C 180.000} C_DIS
LIN {X 152.500,Y 82.490,Z 52.000,A 180.000,B 0.000,C 180.000} C_DIS
LIN {X 152.331,Y 82.490,Z 52.000,A 180.000,B 0.000,C 180.000} C_DIS
LIN {X 152.331,Y 82.490,Z 57.000,A 180.000,B 0.000,C 180.000} C_DIS
LIN {X 141.045,Y 82.490,Z 57.000,A 180.000,B 0.000,C 180.000} C_DIS
LIN {X 141.045,Y 82.490,Z 62.000,A 180.000,B 0.000,C 180.000} C_DIS
LIN {X 83.093,Y 82.490,Z 62.000,A 180.000,B 0.000,C 180.000} C_DIS
LIN {X 83.093,Y 82.490,Z 57.000,A 180.000,B 0.000,C 180.000} C_DIS
LIN {X 71.907,Y 82.490,Z 57.000,A 180.000,B 0.000,C 180.000} C_DIS
LIN {X 71.905,Y 82.490,Z 62.000,A 180.000,B 0.000,C 180.000} C_DIS
LIN {X 13.955,Y 82.490,Z 62.000,A 180.000,B 0.000,C 180.000} C_DIS
LIN {X 13.955,Y 82.490,Z 57.000,A 180.000,B 0.000,C 180.000} C_DIS
LIN {X 2.669,Y 82.490,Z 57.000,A 180.000,B 0.000,C 180.000} C_DIS
LIN {X 2.669,Y 82.490,Z 52.000,A 180.000,B 0.000,C 180.000} C_DIS
LIN {X 2.500,Y 82.490,Z 52.000,A 180.000,B 0.000,C 180.000} C_DIS
LIN {X 2.500,Y 82.490,Z 45.000,A 180.000,B 0.000,C 180.000} C_DIS
LIN {X -0.010,Y 82.490,Z 45.000,A 180.000,B 0.000,C 180.000} C_DIS
; Link Move Starts
LIN {X -0.120,Y 82.490,Z 45.026,A 180.000,B 0.000,C 180.000} C_DIS
LIN {X -0.230,Y 82.490,Z 45.051,A 180.000,B 0.000,C 180.000} C_DIS
LIN {X -0.771,Y 82.803,Z 45.051,A 180.000,B 0.000,C 180.000} C_DIS
LIN {X -0.771,Y 83.427,Z 45.051,A 180.000,B 0.000,C 180.000} C_DIS
LIN {X -0.230,Y 83.740,Z 45.051,A 180.000,B 0.000,C 180.000} C_DIS
LIN {X -0.120,Y 83.740,Z 45.026,A 180.000,B 0.000,C 180.000} C_DIS
LIN {X -0.010,Y 83.740,Z 45.000,A 180.000,B 0.000,C 180.000} C_DIS
; Cutting Move Starts
LIN {X 2.500,Y 83.740,Z 45.000,A 180.000,B 0.000,C 180.000} C_DIS
LIN {X 2.500,Y 83.740,Z 52.000,A 180.000,B 0.000,C 180.000} C_DIS
LIN {X 2.762,Y 83.740,Z 52.000,A 180.000,B 0.000,C 180.000} C_DIS
LIN {X 2.765,Y 83.740,Z 57.000,A 180.000,B 0.000,C 180.000} C_DIS
LIN {X 15.204,Y 83.740,Z 57.000,A 180.000,B 0.000,C 180.000} C_DIS
LIN {X 15.204,Y 83.740,Z 62.000,A 180.000,B 0.000,C 180.000} C_DIS
LIN {X 73.347,Y 83.740,Z 62.000,A 180.000,B 0.000,C 180.000} C_DIS
LIN {X 73.347,Y 83.740,Z 57.000,A 180.000,B 0.000,C 180.000} C_DIS
LIN {X 81.653,Y 83.740,Z 57.000,A 180.000,B 0.000,C 180.000} C_DIS
LIN {X 81.653,Y 83.740,Z 62.000,A 180.000,B 0.000,C 180.000} C_DIS
LIN {X 91.534,Y 83.740,Z 62.000,A 180.000,B 0.000,C 180.000} C_DIS
LIN {X 91.538,Y 83.740,Z 67.555,A 180.000,B 0.000,C 180.000} C_DIS
LIN {X 91.793,Y 83.740,Z 67.776,A 180.000,B 0.000,C 180.000} C_DIS
LIN {X 92.677,Y 83.740,Z 68.453,A 180.000,B 0.000,C 180.000} C_DIS
LIN {X 93.537,Y 83.740,Z 69.014,A 180.000,B 0.000,C 180.000} C_DIS
LIN {X 94.335,Y 83.740,Z 69.443,A 180.000,B 0.000,C 180.000} C_DIS
LIN {X 94.608,Y 83.740,Z 69.561,A 180.000,B 0.000,C 180.000} C_DIS
LIN {X 95.176,Y 83.740,Z 69.796,A 180.000,B 0.000,C 180.000} C_DIS
LIN {X 95.943,Y 83.740,Z 70.026,A 180.000,B 0.000,C 180.000} C_DIS
LIN {X 96.446,Y 83.740,Z 70.119,A 180.000,B 0.000,C 180.000} C_DIS
LIN {X 96.740,Y 83.740,Z 70.168,A 180.000,B 0.000,C 180.000} C_DIS
LIN {X 97.295,Y 83.740,Z 70.204,A 180.000,B 0.000,C 180.000} C_DIS
LIN {X 97.539,Y 83.740,Z 70.213,A 180.000,B 0.000,C 180.000} C_DIS
LIN {X 98.126,Y 83.740,Z 70.178,A 180.000,B 0.000,C 180.000} C_DIS
LIN {X 98.307,Y 83.740,Z 70.162,A 180.000,B 0.000,C 180.000} C_DIS
LIN {X 99.047,Y 83.740,Z 70.028,A 180.000,B 0.000,C 180.000} C_DIS
LIN {X 99.453,Y 83.740,Z 69.909,A 180.000,B 0.000,C 180.000} C_DIS
LIN {X 99.837,Y 83.740,Z 69.791,A 180.000,B 0.000,C 180.000} C_DIS
LIN {X 100.644,Y 83.740,Z 69.453,A 180.000,B 0.000,C 180.000} C_DIS
LIN {X 101.454,Y 83.740,Z 69.020,A 180.000,B 0.000,C 180.000} C_DIS
LIN {X 102.308,Y 83.740,Z 68.464,A 180.000,B 0.000,C 180.000} C_DIS
LIN {X 103.138,Y 83.740,Z 67.832,A 180.000,B 0.000,C 180.000} C_DIS
LIN {X 103.462,Y 83.740,Z 67.555,A 180.000,B 0.000,C 180.000} C_DIS
LIN {X 103.462,Y 83.740,Z 62.000,A 180.000,B 0.000,C 180.000} C_DIS
LIN {X 139.792,Y 83.740,Z 62.000,A 180.000,B 0.000,C 180.000} C_DIS
LIN {X 139.796,Y 83.740,Z 57.000,A 180.000,B 0.000,C 180.000} C_DIS
LIN {X 152.235,Y 83.740,Z 57.000,A 180.000,B 0.000,C 180.000} C_DIS
LIN {X 152.235,Y 83.740,Z 52.000,A 180.000,B 0.000,C 180.000} C_DIS
LIN {X 152.500,Y 83.740,Z 52.000,A 180.000,B 0.000,C 180.000} C_DIS
LIN {X 152.500,Y 83.740,Z 45.000,A 180.000,B 0.000,C 180.000} C_DIS
LIN {X 155.010,Y 83.740,Z 45.000,A 180.000,B 0.000,C 180.000} C_DIS
; Link Move Starts
LIN {X 155.120,Y 83.740,Z 45.026,A 180.000,B 0.000,C 180.000} C_DIS
LIN {X 155.230,Y 83.740,Z 45.051,A 180.000,B 0.000,C 180.000} C_DIS
LIN {X 155.771,Y 84.052,Z 45.051,A 180.000,B 0.000,C 180.000} C_DIS
LIN {X 155.771,Y 84.677,Z 45.051,A 180.000,B 0.000,C 180.000} C_DIS
LIN {X 155.230,Y 84.990,Z 45.051,A 180.000,B 0.000,C 180.000} C_DIS
LIN {X 155.120,Y 84.990,Z 45.026,A 180.000,B 0.000,C 180.000} C_DIS
LIN {X 155.010,Y 84.990,Z 45.000,A 180.000,B 0.000,C 180.000} C_DIS
; Cutting Move Starts
LIN {X 152.500,Y 84.990,Z 45.000,A 180.000,B 0.000,C 180.000} C_DIS
LIN {X 152.500,Y 84.990,Z 52.000,A 180.000,B 0.000,C 180.000} C_DIS
LIN {X 152.121,Y 84.990,Z 52.000,A 180.000,B 0.000,C 180.000} C_DIS
LIN {X 152.117,Y 84.990,Z 57.000,A 180.000,B 0.000,C 180.000} C_DIS
LIN {X 138.546,Y 84.990,Z 57.000,A 180.000,B 0.000,C 180.000} C_DIS
LIN {X 138.546,Y 84.990,Z 62.000,A 180.000,B 0.000,C 180.000} C_DIS
LIN {X 105.768,Y 84.990,Z 62.000,A 180.000,B 0.000,C 180.000} C_DIS
LIN {X 105.765,Y 84.990,Z 67.558,A 180.000,B 0.000,C 180.000} C_DIS
LIN {X 105.326,Y 84.990,Z 68.077,A 180.000,B 0.000,C 180.000} C_DIS
LIN {X 104.395,Y 84.990,Z 69.089,A 180.000,B 0.000,C 180.000} C_DIS
LIN {X 103.527,Y 84.990,Z 69.943,A 180.000,B 0.000,C 180.000} C_DIS
LIN {X 102.677,Y 84.990,Z 70.688,A 180.000,B 0.000,C 180.000} C_DIS
LIN {X 101.889,Y 84.990,Z 71.291,A 180.000,B 0.000,C 180.000} C_DIS
LIN {X 101.083,Y 84.990,Z 71.815,A 180.000,B 0.000,C 180.000} C_DIS
LIN {X 100.367,Y 84.990,Z 72.198,A 180.000,B 0.000,C 180.000} C_DIS
LIN {X 99.625,Y 84.990,Z 72.509,A 180.000,B 0.000,C 180.000} C_DIS
LIN {X 99.387,Y 84.990,Z 72.584,A 180.000,B 0.000,C 180.000} C_DIS
LIN {X 98.915,Y 84.990,Z 72.723,A 180.000,B 0.000,C 180.000} C_DIS
LIN {X 98.249,Y 84.990,Z 72.843,A 180.000,B 0.000,C 180.000} C_DIS
LIN {X 98.008,Y 84.990,Z 72.866,A 180.000,B 0.000,C 180.000} C_DIS
LIN {X 97.516,Y 84.990,Z 72.894,A 180.000,B 0.000,C 180.000} C_DIS
LIN {X 96.877,Y 84.990,Z 72.859,A 180.000,B 0.000,C 180.000} C_DIS
LIN {X 96.662,Y 84.990,Z 72.829,A 180.000,B 0.000,C 180.000} C_DIS
LIN {X 96.077,Y 84.990,Z 72.721,A 180.000,B 0.000,C 180.000} C_DIS
LIN {X 95.401,Y 84.990,Z 72.518,A 180.000,B 0.000,C 180.000} C_DIS
LIN {X 94.977,Y 84.990,Z 72.344,A 180.000,B 0.000,C 180.000} C_DIS
LIN {X 94.618,Y 84.990,Z 72.192,A 180.000,B 0.000,C 180.000} C_DIS
LIN {X 93.907,Y 84.990,Z 71.810,A 180.000,B 0.000,C 180.000} C_DIS
LIN {X 93.108,Y 84.990,Z 71.289,A 180.000,B 0.000,C 180.000} C_DIS
LIN {X 92.317,Y 84.990,Z 70.683,A 180.000,B 0.000,C 180.000} C_DIS
LIN {X 91.474,Y 84.990,Z 69.943,A 180.000,B 0.000,C 180.000} C_DIS
LIN {X 90.588,Y 84.990,Z 69.071,A 180.000,B 0.000,C 180.000} C_DIS
LIN {X 89.625,Y 84.990,Z 68.022,A 180.000,B 0.000,C 180.000} C_DIS
LIN {X 89.232,Y 84.990,Z 67.555,A 180.000,B 0.000,C 180.000} C_DIS
LIN {X 89.230,Y 84.990,Z 62.000,A 180.000,B 0.000,C 180.000} C_DIS
LIN {X 77.783,Y 84.990,Z 62.000,A 180.000,B 0.000,C 180.000} C_DIS
LIN {X 77.783,Y 84.990,Z 57.000,A 180.000,B 0.000,C 180.000} C_DIS
LIN {X 77.217,Y 84.990,Z 57.000,A 180.000,B 0.000,C 180.000} C_DIS
LIN {X 77.217,Y 84.990,Z 62.000,A 180.000,B 0.000,C 180.000} C_DIS
LIN {X 16.454,Y 84.990,Z 62.000,A 180.000,B 0.000,C 180.000} C_DIS
LIN {X 16.454,Y 84.990,Z 57.000,A 180.000,B 0.000,C 180.000} C_DIS
LIN {X 2.879,Y 84.990,Z 57.000,A 180.000,B 0.000,C 180.000} C_DIS
LIN {X 2.879,Y 84.990,Z 52.000,A 180.000,B 0.000,C 180.000} C_DIS
LIN {X 2.500,Y 84.990,Z 52.000,A 180.000,B 0.000,C 180.000} C_DIS
LIN {X 2.500,Y 84.990,Z 45.000,A 180.000,B 0.000,C 180.000} C_DIS
LIN {X -0.010,Y 84.990,Z 45.000,A 180.000,B 0.000,C 180.000} C_DIS
; Link Move Starts
LIN {X -0.120,Y 84.990,Z 45.026,A 180.000,B 0.000,C 180.000} C_DIS
LIN {X -0.230,Y 84.990,Z 45.051,A 180.000,B 0.000,C 180.000} C_DIS
LIN {X -0.771,Y 85.302,Z 45.051,A 180.000,B 0.000,C 180.000} C_DIS
LIN {X -0.771,Y 85.927,Z 45.051,A 180.000,B 0.000,C 180.000} C_DIS
LIN {X -0.230,Y 86.240,Z 45.051,A 180.000,B 0.000,C 180.000} C_DIS
LIN {X -0.120,Y 86.240,Z 45.026,A 180.000,B 0.000,C 180.000} C_DIS
LIN {X -0.010,Y 86.240,Z 45.000,A 180.000,B 0.000,C 180.000} C_DIS
; Cutting Move Starts
LIN {X 2.500,Y 86.240,Z 45.000,A 180.000,B 0.000,C 180.000} C_DIS
LIN {X 2.500,Y 86.240,Z 52.000,A 180.000,B 0.000,C 180.000} C_DIS
LIN {X 3.011,Y 86.240,Z 52.000,A 180.000,B 0.000,C 180.000} C_DIS
LIN {X 3.011,Y 86.240,Z 57.000,A 180.000,B 0.000,C 180.000} C_DIS
LIN {X 17.704,Y 86.240,Z 57.000,A 180.000,B 0.000,C 180.000} C_DIS
LIN {X 17.704,Y 86.240,Z 62.000,A 180.000,B 0.000,C 180.000} C_DIS
LIN {X 87.592,Y 86.240,Z 62.000,A 180.000,B 0.000,C 180.000} C_DIS
LIN {X 87.593,Y 86.240,Z 67.555,A 180.000,B 0.000,C 180.000} C_DIS
LIN {X 88.499,Y 86.240,Z 68.807,A 180.000,B 0.000,C 180.000} C_DIS
LIN {X 89.448,Y 86.240,Z 70.035,A 180.000,B 0.000,C 180.000} C_DIS
LIN {X 89.763,Y 86.240,Z 70.417,A 180.000,B 0.000,C 180.000} C_DIS
LIN {X 90.436,Y 86.240,Z 71.214,A 180.000,B 0.000,C 180.000} C_DIS
LIN {X 91.254,Y 86.240,Z 72.109,A 180.000,B 0.000,C 180.000} C_DIS
LIN {X 91.790,Y 86.240,Z 72.640,A 180.000,B 0.000,C 180.000} C_DIS
LIN {X 92.083,Y 86.240,Z 72.923,A 180.000,B 0.000,C 180.000} C_DIS
LIN {X 92.650,Y 86.240,Z 73.424,A 180.000,B 0.000,C 180.000} C_DIS
LIN {X 92.896,Y 86.240,Z 73.634,A 180.000,B 0.000,C 180.000} C_DIS
LIN {X 93.541,Y 86.240,Z 74.124,A 180.000,B 0.000,C 180.000} C_DIS
LIN {X 94.276,Y 86.240,Z 74.604,A 180.000,B 0.000,C 180.000} C_DIS
LIN {X 94.892,Y 86.240,Z 74.935,A 180.000,B 0.000,C 180.000} C_DIS
LIN {X 95.204,Y 86.240,Z 75.068,A 180.000,B 0.000,C 180.000} C_DIS
LIN {X 95.625,Y 86.240,Z 75.241,A 180.000,B 0.000,C 180.000} C_DIS
LIN {X 96.214,Y 86.240,Z 75.418,A 180.000,B 0.000,C 180.000} C_DIS
LIN {X 96.683,Y 86.240,Z 75.505,A 180.000,B 0.000,C 180.000} C_DIS
LIN {X 96.916,Y 86.240,Z 75.540,A 180.000,B 0.000,C 180.000} C_DIS
LIN {X 97.369,Y 86.240,Z 75.569,A 180.000,B 0.000,C 180.000} C_DIS
LIN {X 97.543,Y 86.240,Z 75.574,A 180.000,B 0.000,C 180.000} C_DIS
LIN {X 98.004,Y 86.240,Z 75.547,A 180.000,B 0.000,C 180.000} C_DIS
LIN {X 98.211,Y 86.240,Z 75.522,A 180.000,B 0.000,C 180.000} C_DIS
LIN {X 98.776,Y 86.240,Z 75.420,A 180.000,B 0.000,C 180.000} C_DIS
LIN {X 99.197,Y 86.240,Z 75.296,A 180.000,B 0.000,C 180.000} C_DIS
LIN {X 99.403,Y 86.240,Z 75.230,A 180.000,B 0.000,C 180.000} C_DIS
LIN {X 100.069,Y 86.240,Z 74.953,A 180.000,B 0.000,C 180.000} C_DIS
LIN {X 100.320,Y 86.240,Z 74.823,A 180.000,B 0.000,C 180.000} C_DIS
LIN {X 100.733,Y 86.240,Z 74.599,A 180.000,B 0.000,C 180.000} C_DIS
LIN {X 101.464,Y 86.240,Z 74.121,A 180.000,B 0.000,C 180.000} C_DIS
LIN {X 102.130,Y 86.240,Z 73.613,A 180.000,B 0.000,C 180.000} C_DIS
LIN {X 102.545,Y 86.240,Z 73.253,A 180.000,B 0.000,C 180.000} C_DIS
LIN {X 102.942,Y 86.240,Z 72.901,A 180.000,B 0.000,C 180.000} C_DIS
LIN {X 103.682,Y 86.240,Z 72.174,A 180.000,B 0.000,C 180.000} C_DIS
LIN {X 104.012,Y 86.240,Z 71.820,A 180.000,B 0.000,C 180.000} C_DIS
LIN {X 104.577,Y 86.240,Z 71.200,A 180.000,B 0.000,C 180.000} C_DIS
LIN {X 105.468,Y 86.240,Z 70.141,A 180.000,B 0.000,C 180.000} C_DIS
LIN {X 106.443,Y 86.240,Z 68.885,A 180.000,B 0.000,C 180.000} C_DIS
LIN {X 107.405,Y 86.240,Z 67.558,A 180.000,B 0.000,C 180.000} C_DIS
LIN {X 107.407,Y 86.240,Z 62.000,A 180.000,B 0.000,C 180.000} C_DIS
LIN {X 137.296,Y 86.240,Z 62.000,A 180.000,B 0.000,C 180.000} C_DIS
LIN {X 137.296,Y 86.240,Z 57.000,A 180.000,B 0.000,C 180.000} C_DIS
LIN {X 151.989,Y 86.240,Z 57.000,A 180.000,B 0.000,C 180.000} C_DIS
LIN {X 151.989,Y 86.240,Z 52.000,A 180.000,B 0.000,C 180.000} C_DIS
LIN {X 152.500,Y 86.240,Z 52.000,A 180.000,B 0.000,C 180.000} C_DIS
LIN {X 152.500,Y 86.240,Z 45.000,A 180.000,B 0.000,C 180.000} C_DIS
LIN {X 155.010,Y 86.240,Z 45.000,A 180.000,B 0.000,C 180.000} C_DIS
; Link Move Starts
LIN {X 155.120,Y 86.240,Z 45.026,A 180.000,B 0.000,C 180.000} C_DIS
LIN {X 155.230,Y 86.240,Z 45.051,A 180.000,B 0.000,C 180.000} C_DIS
LIN {X 155.771,Y 86.552,Z 45.051,A 180.000,B 0.000,C 180.000} C_DIS
LIN {X 155.771,Y 87.177,Z 45.051,A 180.000,B 0.000,C 180.000} C_DIS
LIN {X 155.230,Y 87.490,Z 45.051,A 180.000,B 0.000,C 180.000} C_DIS
LIN {X 155.120,Y 87.490,Z 45.026,A 180.000,B 0.000,C 180.000} C_DIS
LIN {X 155.010,Y 87.490,Z 45.000,A 180.000,B 0.000,C 180.000} C_DIS
; Cutting Move Starts
LIN {X 152.500,Y 87.490,Z 45.000,A 180.000,B 0.000,C 180.000} C_DIS
LIN {X 152.500,Y 87.490,Z 52.000,A 180.000,B 0.000,C 180.000} C_DIS
LIN {X 151.828,Y 87.490,Z 52.000,A 180.000,B 0.000,C 180.000} C_DIS
LIN {X 151.827,Y 87.490,Z 57.000,A 180.000,B 0.000,C 180.000} C_DIS
LIN {X 136.046,Y 87.490,Z 57.000,A 180.000,B 0.000,C 180.000} C_DIS
LIN {X 136.046,Y 87.490,Z 62.000,A 180.000,B 0.000,C 180.000} C_DIS
LIN {X 108.671,Y 87.490,Z 62.000,A 180.000,B 0.000,C 180.000} C_DIS
LIN {X 108.668,Y 87.490,Z 67.559,A 180.000,B 0.000,C 180.000} C_DIS
LIN {X 107.461,Y 87.490,Z 69.437,A 180.000,B 0.000,C 180.000} C_DIS
LIN {X 106.423,Y 87.490,Z 70.964,A 180.000,B 0.000,C 180.000} C_DIS
LIN {X 105.441,Y 87.490,Z 72.320,A 180.000,B 0.000,C 180.000} C_DIS
LIN {X 104.587,Y 87.490,Z 73.420,A 180.000,B 0.000,C 180.000} C_DIS
LIN {X 103.818,Y 87.490,Z 74.333,A 180.000,B 0.000,C 180.000} C_DIS
LIN {X 103.518,Y 87.490,Z 74.668,A 180.000,B 0.000,C 180.000} C_DIS
LIN {X 103.004,Y 87.490,Z 75.224,A 180.000,B 0.000,C 180.000} C_DIS
LIN {X 102.362,Y 87.490,Z 75.854,A 180.000,B 0.000,C 180.000} C_DIS
LIN {X 102.007,Y 87.490,Z 76.172,A 180.000,B 0.000,C 180.000} C_DIS
LIN {X 101.605,Y 87.490,Z 76.520,A 180.000,B 0.000,C 180.000} C_DIS
LIN {X 101.037,Y 87.490,Z 76.952,A 180.000,B 0.000,C 180.000} C_DIS
LIN {X 100.372,Y 87.490,Z 77.388,A 180.000,B 0.000,C 180.000} C_DIS
LIN {X 100.100,Y 87.490,Z 77.537,A 180.000,B 0.000,C 180.000} C_DIS
LIN {X 99.800,Y 87.490,Z 77.695,A 180.000,B 0.000,C 180.000} C_DIS
LIN {X 99.208,Y 87.490,Z 77.941,A 180.000,B 0.000,C 180.000} C_DIS
LIN {X 99.025,Y 87.490,Z 78.003,A 180.000,B 0.000,C 180.000} C_DIS
LIN {X 98.640,Y 87.490,Z 78.116,A 180.000,B 0.000,C 180.000} C_DIS
LIN {X 98.146,Y 87.490,Z 78.205,A 180.000,B 0.000,C 180.000} C_DIS
LIN {X 97.922,Y 87.490,Z 78.232,A 180.000,B 0.000,C 180.000} C_DIS
LIN {X 97.490,Y 87.490,Z 78.255,A 180.000,B 0.000,C 180.000} C_DIS
LIN {X 97.009,Y 87.490,Z 78.226,A 180.000,B 0.000,C 180.000} C_DIS
LIN {X 96.742,Y 87.490,Z 78.187,A 180.000,B 0.000,C 180.000} C_DIS
LIN {X 96.348,Y 87.490,Z 78.113,A 180.000,B 0.000,C 180.000} C_DIS
LIN {X 95.852,Y 87.490,Z 77.964,A 180.000,B 0.000,C 180.000} C_DIS
LIN {X 95.432,Y 87.490,Z 77.793,A 180.000,B 0.000,C 180.000} C_DIS
LIN {X 95.164,Y 87.490,Z 77.678,A 180.000,B 0.000,C 180.000} C_DIS
LIN {X 94.645,Y 87.490,Z 77.399,A 180.000,B 0.000,C 180.000} C_DIS
LIN {X 93.971,Y 87.490,Z 76.959,A 180.000,B 0.000,C 180.000} C_DIS
LIN {X 93.580,Y 87.490,Z 76.663,A 180.000,B 0.000,C 180.000} C_DIS
LIN {X 93.331,Y 87.490,Z 76.467,A 180.000,B 0.000,C 180.000} C_DIS
LIN {X 92.720,Y 87.490,Z 75.929,A 180.000,B 0.000,C 180.000} C_DIS
LIN {X 92.454,Y 87.490,Z 75.677,A 180.000,B 0.000,C 180.000} C_DIS
LIN {X 91.944,Y 87.490,Z 75.171,A 180.000,B 0.000,C 180.000} C_DIS
LIN {X 91.242,Y 87.490,Z 74.402,A 180.000,B 0.000,C 180.000} C_DIS
LIN {X 90.864,Y 87.490,Z 73.958,A 180.000,B 0.000,C 180.000} C_DIS
LIN {X 90.353,Y 87.490,Z 73.345,A 180.000,B 0.000,C 180.000} C_DIS
LIN {X 89.519,Y 87.490,Z 72.266,A 180.000,B 0.000,C 180.000} C_DIS
LIN {X 88.512,Y 87.490,Z 70.871,A 180.000,B 0.000,C 180.000} C_DIS
LIN {X 87.461,Y 87.490,Z 69.319,A 180.000,B 0.000,C 180.000} C_DIS
LIN {X 86.329,Y 87.490,Z 67.555,A 180.000,B 0.000,C 180.000} C_DIS
LIN {X 86.328,Y 87.490,Z 62.000,A 180.000,B 0.000,C 180.000} C_DIS
LIN {X 18.954,Y 87.490,Z 62.000,A 180.000,B 0.000,C 180.000} C_DIS
LIN {X 18.954,Y 87.490,Z 57.000,A 180.000,B 0.000,C 180.000} C_DIS
LIN {X 3.172,Y 87.490,Z 57.000,A 180.000,B 0.000,C 180.000} C_DIS
LIN {X 3.172,Y 87.490,Z 52.000,A 180.000,B 0.000,C 180.000} C_DIS
LIN {X 2.500,Y 87.490,Z 52.000,A 180.000,B 0.000,C 180.000} C_DIS
LIN {X 2.499,Y 87.490,Z 45.000,A 180.000,B 0.000,C 180.000} C_DIS
LIN {X -0.010,Y 87.490,Z 45.000,A 180.000,B 0.000,C 180.000} C_DIS
; Link Move Starts
LIN {X -0.120,Y 87.490,Z 45.026,A 180.000,B 0.000,C 180.000} C_DIS
LIN {X -0.230,Y 87.490,Z 45.051,A 180.000,B 0.000,C 180.000} C_DIS
LIN {X -0.771,Y 87.802,Z 45.051,A 180.000,B 0.000,C 180.000} C_DIS
LIN {X -0.771,Y 88.427,Z 45.051,A 180.000,B 0.000,C 180.000} C_DIS
LIN {X -0.230,Y 88.740,Z 45.051,A 180.000,B 0.000,C 180.000} C_DIS
LIN {X -0.120,Y 88.740,Z 45.026,A 180.000,B 0.000,C 180.000} C_DIS
LIN {X -0.010,Y 88.740,Z 45.000,A 180.000,B 0.000,C 180.000} C_DIS
; Cutting Move Starts
LIN {X 2.500,Y 88.740,Z 45.000,A 180.000,B 0.000,C 180.000} C_DIS
LIN {X 2.500,Y 88.740,Z 52.000,A 180.000,B 0.000,C 180.000} C_DIS
LIN {X 3.352,Y 88.740,Z 52.000,A 180.000,B 0.000,C 180.000} C_DIS
LIN {X 3.352,Y 88.740,Z 57.000,A 180.000,B 0.000,C 180.000} C_DIS
LIN {X 20.204,Y 88.740,Z 57.000,A 180.000,B 0.000,C 180.000} C_DIS
LIN {X 20.204,Y 88.740,Z 62.000,A 180.000,B 0.000,C 180.000} C_DIS
LIN {X 85.324,Y 88.740,Z 62.000,A 180.000,B 0.000,C 180.000} C_DIS
LIN {X 85.326,Y 88.740,Z 67.555,A 180.000,B 0.000,C 180.000} C_DIS
LIN {X 86.470,Y 88.740,Z 69.515,A 180.000,B 0.000,C 180.000} C_DIS
LIN {X 87.628,Y 88.740,Z 71.418,A 180.000,B 0.000,C 180.000} C_DIS
LIN {X 88.728,Y 88.740,Z 73.136,A 180.000,B 0.000,C 180.000} C_DIS
LIN {X 89.617,Y 88.740,Z 74.449,A 180.000,B 0.000,C 180.000} C_DIS
LIN {X 90.535,Y 88.740,Z 75.720,A 180.000,B 0.000,C 180.000} C_DIS
LIN {X 91.231,Y 88.740,Z 76.620,A 180.000,B 0.000,C 180.000} C_DIS
LIN {X 91.693,Y 88.740,Z 77.175,A 180.000,B 0.000,C 180.000} C_DIS
LIN {X 92.052,Y 88.740,Z 77.595,A 180.000,B 0.000,C 180.000} C_DIS
LIN {X 92.635,Y 88.740,Z 78.233,A 180.000,B 0.000,C 180.000} C_DIS
LIN {X 93.091,Y 88.740,Z 78.686,A 180.000,B 0.000,C 180.000} C_DIS
LIN {X 93.345,Y 88.740,Z 78.924,A 180.000,B 0.000,C 180.000} C_DIS
LIN {X 93.849,Y 88.740,Z 79.368,A 180.000,B 0.000,C 180.000} C_DIS
LIN {X 94.084,Y 88.740,Z 79.554,A 180.000,B 0.000,C 180.000} C_DIS
LIN {X 94.400,Y 88.740,Z 79.792,A 180.000,B 0.000,C 180.000} C_DIS
LIN {X 95.011,Y 88.740,Z 80.191,A 180.000,B 0.000,C 180.000} C_DIS
LIN {X 95.420,Y 88.740,Z 80.412,A 180.000,B 0.000,C 180.000} C_DIS
LIN {X 95.629,Y 88.740,Z 80.505,A 180.000,B 0.000,C 180.000} C_DIS
LIN {X 96.076,Y 88.740,Z 80.687,A 180.000,B 0.000,C 180.000} C_DIS
LIN {X 96.478,Y 88.740,Z 80.808,A 180.000,B 0.000,C 180.000} C_DIS
LIN {X 96.794,Y 88.740,Z 80.868,A 180.000,B 0.000,C 180.000} C_DIS
LIN {X 97.073,Y 88.740,Z 80.908,A 180.000,B 0.000,C 180.000} C_DIS
LIN {X 97.269,Y 88.740,Z 80.924,A 180.000,B 0.000,C 180.000} C_DIS
LIN {X 97.529,Y 88.740,Z 80.935,A 180.000,B 0.000,C 180.000} C_DIS
LIN {X 97.835,Y 88.740,Z 80.918,A 180.000,B 0.000,C 180.000} C_DIS
LIN {X 98.109,Y 88.740,Z 80.884,A 180.000,B 0.000,C 180.000} C_DIS
LIN {X 98.495,Y 88.740,Z 80.815,A 180.000,B 0.000,C 180.000} C_DIS
LIN {X 98.795,Y 88.740,Z 80.728,A 180.000,B 0.000,C 180.000} C_DIS
LIN {X 98.994,Y 88.740,Z 80.660,A 180.000,B 0.000,C 180.000} C_DIS
LIN {X 99.512,Y 88.740,Z 80.445,A 180.000,B 0.000,C 180.000} C_DIS
LIN {X 99.739,Y 88.740,Z 80.328,A 180.000,B 0.000,C 180.000} C_DIS
LIN {X 100.004,Y 88.740,Z 80.182,A 180.000,B 0.000,C 180.000} C_DIS
LIN {X 100.613,Y 88.740,Z 79.783,A 180.000,B 0.000,C 180.000} C_DIS
LIN {X 101.079,Y 88.740,Z 79.428,A 180.000,B 0.000,C 180.000} C_DIS
LIN {X 101.420,Y 88.740,Z 79.133,A 180.000,B 0.000,C 180.000} C_DIS
LIN {X 101.779,Y 88.740,Z 78.811,A 180.000,B 0.000,C 180.000} C_DIS
LIN {X 102.308,Y 88.740,Z 78.292,A 180.000,B 0.000,C 180.000} C_DIS
LIN {X 102.754,Y 88.740,Z 77.809,A 180.000,B 0.000,C 180.000} C_DIS
LIN {X 103.062,Y 88.740,Z 77.465,A 180.000,B 0.000,C 180.000} C_DIS
LIN {X 103.705,Y 88.740,Z 76.700,A 180.000,B 0.000,C 180.000} C_DIS
LIN {X 104.437,Y 88.740,Z 75.758,A 180.000,B 0.000,C 180.000} C_DIS
LIN {X 105.319,Y 88.740,Z 74.540,A 180.000,B 0.000,C 180.000} C_DIS
LIN {X 106.190,Y 88.740,Z 73.260,A 180.000,B 0.000,C 180.000} C_DIS
LIN {X 107.282,Y 88.740,Z 71.561,A 180.000,B 0.000,C 180.000} C_DIS
LIN {X 108.423,Y 88.740,Z 69.695,A 180.000,B 0.000,C 180.000} C_DIS
LIN {X 109.672,Y 88.740,Z 67.559,A 180.000,B 0.000,C 180.000} C_DIS
LIN {X 109.674,Y 88.740,Z 62.000,A 180.000,B 0.000,C 180.000} C_DIS
LIN {X 134.796,Y 88.740,Z 62.000,A 180.000,B 0.000,C 180.000} C_DIS
LIN {X 134.796,Y 88.740,Z 57.000,A 180.000,B 0.000,C 180.000} C_DIS
LIN {X 151.648,Y 88.740,Z 57.000,A 180.000,B 0.000,C 180.000} C_DIS
LIN {X 151.648,Y 88.740,Z 52.000,A 180.000,B 0.000,C 180.000} C_DIS
LIN {X 152.500,Y 88.740,Z 52.000,A 180.000,B 0.000,C 180.000} C_DIS
LIN {X 152.500,Y 88.740,Z 45.000,A 180.000,B 0.000,C 180.000} C_DIS
LIN {X 155.010,Y 88.740,Z 45.000,A 180.000,B 0.000,C 180.000} C_DIS
; Link Move Starts
LIN {X 155.120,Y 88.740,Z 45.026,A 180.000,B 0.000,C 180.000} C_DIS
LIN {X 155.230,Y 88.740,Z 45.051,A 180.000,B 0.000,C 180.000} C_DIS
LIN {X 155.771,Y 89.052,Z 45.051,A 180.000,B 0.000,C 180.000} C_DIS
LIN {X 155.771,Y 89.677,Z 45.051,A 180.000,B 0.000,C 180.000} C_DIS
LIN {X 155.230,Y 89.989,Z 45.051,A 180.000,B 0.000,C 180.000} C_DIS
LIN {X 155.120,Y 89.989,Z 45.026,A 180.000,B 0.000,C 180.000} C_DIS
LIN {X 155.010,Y 89.989,Z 45.000,A 180.000,B 0.000,C 180.000} C_DIS
; Cutting Move Starts
LIN {X 152.500,Y 89.989,Z 45.000,A 180.000,B 0.000,C 180.000} C_DIS
LIN {X 152.500,Y 89.989,Z 52.000,A 180.000,B 0.000,C 180.000} C_DIS
LIN {X 151.451,Y 89.989,Z 52.000,A 180.000,B 0.000,C 180.000} C_DIS
LIN {X 151.450,Y 89.989,Z 57.000,A 180.000,B 0.000,C 180.000} C_DIS
LIN {X 133.546,Y 89.989,Z 57.000,A 180.000,B 0.000,C 180.000} C_DIS
LIN {X 133.544,Y 89.989,Z 62.000,A 180.000,B 0.000,C 180.000} C_DIS
LIN {X 110.479,Y 89.989,Z 62.000,A 180.000,B 0.000,C 180.000} C_DIS
LIN {X 110.479,Y 89.989,Z 67.555,A 180.000,B 0.000,C 180.000} C_DIS
LIN {X 109.373,Y 89.989,Z 69.594,A 180.000,B 0.000,C 180.000} C_DIS
LIN {X 108.070,Y 89.989,Z 71.914,A 180.000,B 0.000,C 180.000} C_DIS
LIN {X 106.849,Y 89.989,Z 74.005,A 180.000,B 0.000,C 180.000} C_DIS
LIN {X 105.908,Y 89.989,Z 75.543,A 180.000,B 0.000,C 180.000} C_DIS
LIN {X 104.921,Y 89.989,Z 77.079,A 180.000,B 0.000,C 180.000} C_DIS
LIN {X 104.211,Y 89.989,Z 78.121,A 180.000,B 0.000,C 180.000} C_DIS
LIN {X 103.427,Y 89.989,Z 79.202,A 180.000,B 0.000,C 180.000} C_DIS
LIN {X 102.826,Y 89.989,Z 79.977,A 180.000,B 0.000,C 180.000} C_DIS
LIN {X 102.299,Y 89.989,Z 80.602,A 180.000,B 0.000,C 180.000} C_DIS
LIN {X 101.981,Y 89.989,Z 80.962,A 180.000,B 0.000,C 180.000} C_DIS
LIN {X 101.610,Y 89.989,Z 81.362,A 180.000,B 0.000,C 180.000} C_DIS
LIN {X 101.192,Y 89.989,Z 81.771,A 180.000,B 0.000,C 180.000} C_DIS
LIN {X 100.805,Y 89.989,Z 82.119,A 180.000,B 0.000,C 180.000} C_DIS
LIN {X 100.544,Y 89.989,Z 82.343,A 180.000,B 0.000,C 180.000} C_DIS
LIN {X 100.186,Y 89.989,Z 82.614,A 180.000,B 0.000,C 180.000} C_DIS
LIN {X 99.629,Y 89.989,Z 82.980,A 180.000,B 0.000,C 180.000} C_DIS
LIN {X 99.323,Y 89.989,Z 83.147,A 180.000,B 0.000,C 180.000} C_DIS
LIN {X 99.127,Y 89.989,Z 83.236,A 180.000,B 0.000,C 180.000} C_DIS
LIN {X 98.679,Y 89.989,Z 83.416,A 180.000,B 0.000,C 180.000} C_DIS
LIN {X 98.371,Y 89.989,Z 83.508,A 180.000,B 0.000,C 180.000} C_DIS
LIN {X 98.063,Y 89.989,Z 83.564,A 180.000,B 0.000,C 180.000} C_DIS
LIN {X 97.768,Y 89.989,Z 83.602,A 180.000,B 0.000,C 180.000} C_DIS
LIN {X 97.535,Y 89.989,Z 83.616,A 180.000,B 0.000,C 180.000} C_DIS
LIN {X 97.246,Y 89.989,Z 83.603,A 180.000,B 0.000,C 180.000} C_DIS
LIN {X 96.900,Y 89.989,Z 83.559,A 180.000,B 0.000,C 180.000} C_DIS
LIN {X 96.618,Y 89.989,Z 83.505,A 180.000,B 0.000,C 180.000} C_DIS
LIN {X 96.302,Y 89.989,Z 83.410,A 180.000,B 0.000,C 180.000} C_DIS
LIN {X 95.827,Y 89.989,Z 83.217,A 180.000,B 0.000,C 180.000} C_DIS
LIN {X 95.613,Y 89.989,Z 83.113,A 180.000,B 0.000,C 180.000} C_DIS
LIN {X 95.363,Y 89.989,Z 82.975,A 180.000,B 0.000,C 180.000} C_DIS
LIN {X 94.802,Y 89.989,Z 82.606,A 180.000,B 0.000,C 180.000} C_DIS
LIN {X 94.410,Y 89.989,Z 82.306,A 180.000,B 0.000,C 180.000} C_DIS
LIN {X 93.986,Y 89.989,Z 81.933,A 180.000,B 0.000,C 180.000} C_DIS
LIN {X 93.696,Y 89.989,Z 81.664,A 180.000,B 0.000,C 180.000} C_DIS
LIN {X 93.321,Y 89.989,Z 81.291,A 180.000,B 0.000,C 180.000} C_DIS
LIN {X 92.861,Y 89.989,Z 80.786,A 180.000,B 0.000,C 180.000} C_DIS
LIN {X 92.482,Y 89.989,Z 80.345,A 180.000,B 0.000,C 180.000} C_DIS
LIN {X 92.105,Y 89.989,Z 79.891,A 180.000,B 0.000,C 180.000} C_DIS
LIN {X 91.551,Y 89.989,Z 79.172,A 180.000,B 0.000,C 180.000} C_DIS
LIN {X 90.756,Y 89.989,Z 78.075,A 180.000,B 0.000,C 180.000} C_DIS
LIN {X 90.002,Y 89.989,Z 76.962,A 180.000,B 0.000,C 180.000} C_DIS
LIN {X 88.997,Y 89.989,Z 75.392,A 180.000,B 0.000,C 180.000} C_DIS
LIN {X 88.049,Y 89.989,Z 73.834,A 180.000,B 0.000,C 180.000} C_DIS
LIN {X 86.853,Y 89.989,Z 71.779,A 180.000,B 0.000,C 180.000} C_DIS
LIN {X 85.485,Y 89.989,Z 69.337,A 180.000,B 0.000,C 180.000} C_DIS
LIN {X 84.521,Y 89.989,Z 67.555,A 180.000,B 0.000,C 180.000} C_DIS
LIN {X 84.521,Y 89.989,Z 62.000,A 180.000,B 0.000,C 180.000} C_DIS
LIN {X 63.489,Y 89.989,Z 62.000,A 180.000,B 0.000,C 180.000} C_DIS
LIN {X 63.489,Y 89.989,Z 66.500,A 180.000,B 0.000,C 180.000} C_DIS
LIN {X 63.363,Y 89.989,Z 66.500,A 180.000,B 0.000,C 180.000} C_DIS
LIN {X 63.363,Y 89.989,Z 70.000,A 180.000,B 0.000,C 180.000} C_DIS
LIN {X 53.637,Y 89.989,Z 70.000,A 180.000,B 0.000,C 180.000} C_DIS
LIN {X 53.637,Y 89.989,Z 66.500,A 180.000,B 0.000,C 180.000} C_DIS
LIN {X 53.511,Y 89.989,Z 66.500,A 180.000,B 0.000,C 180.000} C_DIS
LIN {X 53.511,Y 89.989,Z 62.000,A 180.000,B 0.000,C 180.000} C_DIS
LIN {X 21.454,Y 89.989,Z 62.000,A 180.000,B 0.000,C 180.000} C_DIS
LIN {X 21.454,Y 89.989,Z 57.000,A 180.000,B 0.000,C 180.000} C_DIS
LIN {X 3.550,Y 89.989,Z 57.000,A 180.000,B 0.000,C 180.000} C_DIS
LIN {X 3.549,Y 89.989,Z 52.000,A 180.000,B 0.000,C 180.000} C_DIS
LIN {X 2.500,Y 89.989,Z 52.000,A 180.000,B 0.000,C 180.000} C_DIS
LIN {X 2.500,Y 89.989,Z 45.000,A 180.000,B 0.000,C 180.000} C_DIS
LIN {X -0.010,Y 89.989,Z 45.000,A 180.000,B 0.000,C 180.000} C_DIS
; Link Move Starts
LIN {X -0.120,Y 89.989,Z 45.026,A 180.000,B 0.000,C 180.000} C_DIS
LIN {X -0.230,Y 89.989,Z 45.051,A 180.000,B 0.000,C 180.000} C_DIS
LIN {X -0.771,Y 90.302,Z 45.051,A 180.000,B 0.000,C 180.000} C_DIS
LIN {X -0.771,Y 90.927,Z 45.051,A 180.000,B 0.000,C 180.000} C_DIS
LIN {X -0.230,Y 91.239,Z 45.051,A 180.000,B 0.000,C 180.000} C_DIS
LIN {X -0.120,Y 91.239,Z 45.026,A 180.000,B 0.000,C 180.000} C_DIS
LIN {X -0.010,Y 91.239,Z 45.000,A 180.000,B 0.000,C 180.000} C_DIS
; Cutting Move Starts
LIN {X 2.500,Y 91.239,Z 45.000,A 180.000,B 0.000,C 180.000} C_DIS
LIN {X 2.500,Y 91.239,Z 52.000,A 180.000,B 0.000,C 180.000} C_DIS
LIN {X 3.772,Y 91.239,Z 52.000,A 180.000,B 0.000,C 180.000} C_DIS
LIN {X 3.772,Y 91.239,Z 57.000,A 180.000,B 0.000,C 180.000} C_DIS
LIN {X 22.704,Y 91.239,Z 57.000,A 180.000,B 0.000,C 180.000} C_DIS
LIN {X 22.704,Y 91.239,Z 62.000,A 180.000,B 0.000,C 180.000} C_DIS
LIN {X 51.276,Y 91.239,Z 62.000,A 180.000,B 0.000,C 180.000} C_DIS
LIN {X 51.279,Y 91.239,Z 66.500,A 180.000,B 0.000,C 180.000} C_DIS
LIN {X 51.368,Y 91.239,Z 66.500,A 180.000,B 0.000,C 180.000} C_DIS
LIN {X 51.368,Y 91.239,Z 70.000,A 180.000,B 0.000,C 180.000} C_DIS
LIN {X 65.630,Y 91.239,Z 70.000,A 180.000,B 0.000,C 180.000} C_DIS
LIN {X 65.632,Y 91.239,Z 66.500,A 180.000,B 0.000,C 180.000} C_DIS
LIN {X 65.721,Y 91.239,Z 66.500,A 180.000,B 0.000,C 180.000} C_DIS
LIN {X 65.721,Y 91.239,Z 62.000,A 180.000,B 0.000,C 180.000} C_DIS
LIN {X 83.872,Y 91.239,Z 62.000,A 180.000,B 0.000,C 180.000} C_DIS
LIN {X 83.874,Y 91.239,Z 67.555,A 180.000,B 0.000,C 180.000} C_DIS
LIN {X 84.418,Y 91.239,Z 68.621,A 180.000,B 0.000,C 180.000} C_DIS
LIN {X 86.138,Y 91.239,Z 71.900,A 180.000,B 0.000,C 180.000} C_DIS
LIN {X 87.485,Y 91.239,Z 74.394,A 180.000,B 0.000,C 180.000} C_DIS
LIN {X 88.617,Y 91.239,Z 76.414,A 180.000,B 0.000,C 180.000} C_DIS
LIN {X 89.624,Y 91.239,Z 78.146,A 180.000,B 0.000,C 180.000} C_DIS
LIN {X 90.365,Y 91.239,Z 79.365,A 180.000,B 0.000,C 180.000} C_DIS
LIN {X 91.273,Y 91.239,Z 80.784,A 180.000,B 0.000,C 180.000} C_DIS
LIN {X 91.865,Y 91.239,Z 81.658,A 180.000,B 0.000,C 180.000} C_DIS
LIN {X 92.557,Y 91.239,Z 82.612,A 180.000,B 0.000,C 180.000} C_DIS
LIN {X 92.961,Y 91.239,Z 83.139,A 180.000,B 0.000,C 180.000} C_DIS
LIN {X 93.250,Y 91.239,Z 83.490,A 180.000,B 0.000,C 180.000} C_DIS
LIN {X 93.653,Y 91.239,Z 83.958,A 180.000,B 0.000,C 180.000} C_DIS
LIN {X 93.997,Y 91.239,Z 84.337,A 180.000,B 0.000,C 180.000} C_DIS
LIN {X 94.279,Y 91.239,Z 84.620,A 180.000,B 0.000,C 180.000} C_DIS
LIN {X 94.587,Y 91.239,Z 84.906,A 180.000,B 0.000,C 180.000} C_DIS
LIN {X 94.916,Y 91.239,Z 85.197,A 180.000,B 0.000,C 180.000} C_DIS
LIN {X 95.189,Y 91.239,Z 85.409,A 180.000,B 0.000,C 180.000} C_DIS
LIN {X 95.587,Y 91.239,Z 85.676,A 180.000,B 0.000,C 180.000} C_DIS
LIN {X 95.808,Y 91.239,Z 85.814,A 180.000,B 0.000,C 180.000} C_DIS
LIN {X 96.040,Y 91.239,Z 85.934,A 180.000,B 0.000,C 180.000} C_DIS
LIN {X 96.496,Y 91.239,Z 86.121,A 180.000,B 0.000,C 180.000} C_DIS
LIN {X 96.694,Y 91.239,Z 86.185,A 180.000,B 0.000,C 180.000} C_DIS
LIN {X 96.898,Y 91.239,Z 86.230,A 180.000,B 0.000,C 180.000} C_DIS
LIN {X 97.247,Y 91.239,Z 86.280,A 180.000,B 0.000,C 180.000} C_DIS
LIN {X 97.481,Y 91.239,Z 86.296,A 180.000,B 0.000,C 180.000} C_DIS
LIN {X 97.672,Y 91.239,Z 86.288,A 180.000,B 0.000,C 180.000} C_DIS
LIN {X 97.992,Y 91.239,Z 86.248,A 180.000,B 0.000,C 180.000} C_DIS
LIN {X 98.212,Y 91.239,Z 86.209,A 180.000,B 0.000,C 180.000} C_DIS
LIN {X 98.425,Y 91.239,Z 86.149,A 180.000,B 0.000,C 180.000} C_DIS
LIN {X 98.662,Y 91.239,Z 86.058,A 180.000,B 0.000,C 180.000} C_DIS
LIN {X 98.986,Y 91.239,Z 85.922,A 180.000,B 0.000,C 180.000} C_DIS
LIN {X 99.244,Y 91.239,Z 85.784,A 180.000,B 0.000,C 180.000} C_DIS
LIN {X 99.727,Y 91.239,Z 85.468,A 180.000,B 0.000,C 180.000} C_DIS
LIN {X 99.945,Y 91.239,Z 85.307,A 180.000,B 0.000,C 180.000} C_DIS
LIN {X 100.185,Y 91.239,Z 85.109,A 180.000,B 0.000,C 180.000} C_DIS
LIN {X 100.602,Y 91.239,Z 84.733,A 180.000,B 0.000,C 180.000} C_DIS
LIN {X 100.904,Y 91.239,Z 84.440,A 180.000,B 0.000,C 180.000} C_DIS
LIN {X 101.183,Y 91.239,Z 84.141,A 180.000,B 0.000,C 180.000} C_DIS
LIN {X 101.536,Y 91.239,Z 83.741,A 180.000,B 0.000,C 180.000} C_DIS
LIN {X 101.942,Y 91.239,Z 83.260,A 180.000,B 0.000,C 180.000} C_DIS
LIN {X 102.402,Y 91.239,Z 82.668,A 180.000,B 0.000,C 180.000} C_DIS
LIN {X 103.105,Y 91.239,Z 81.700,A 180.000,B 0.000,C 180.000} C_DIS
LIN {X 103.653,Y 91.239,Z 80.897,A 180.000,B 0.000,C 180.000} C_DIS
LIN {X 104.542,Y 91.239,Z 79.513,A 180.000,B 0.000,C 180.000} C_DIS
LIN {X 105.333,Y 91.239,Z 78.218,A 180.000,B 0.000,C 180.000} C_DIS
LIN {X 106.352,Y 91.239,Z 76.468,A 180.000,B 0.000,C 180.000} C_DIS
LIN {X 107.396,Y 91.239,Z 74.610,A 180.000,B 0.000,C 180.000} C_DIS
LIN {X 108.782,Y 91.239,Z 72.052,A 180.000,B 0.000,C 180.000} C_DIS
LIN {X 110.361,Y 91.239,Z 69.047,A 180.000,B 0.000,C 180.000} C_DIS
LIN {X 111.126,Y 91.239,Z 67.555,A 180.000,B 0.000,C 180.000} C_DIS
LIN {X 111.126,Y 91.239,Z 62.000,A 180.000,B 0.000,C 180.000} C_DIS
LIN {X 132.296,Y 91.239,Z 62.000,A 180.000,B 0.000,C 180.000} C_DIS
LIN {X 132.296,Y 91.239,Z 57.000,A 180.000,B 0.000,C 180.000} C_DIS
LIN {X 151.228,Y 91.239,Z 57.000,A 180.000,B 0.000,C 180.000} C_DIS
LIN {X 151.228,Y 91.239,Z 52.000,A 180.000,B 0.000,C 180.000} C_DIS
LIN {X 152.500,Y 91.239,Z 52.000,A 180.000,B 0.000,C 180.000} C_DIS
LIN {X 152.500,Y 91.239,Z 45.000,A 180.000,B 0.000,C 180.000} C_DIS
LIN {X 155.010,Y 91.239,Z 45.000,A 180.000,B 0.000,C 180.000} C_DIS
; Link Move Starts
LIN {X 155.120,Y 91.239,Z 45.026,A 180.000,B 0.000,C 180.000} C_DIS
LIN {X 155.230,Y 91.239,Z 45.051,A 180.000,B 0.000,C 180.000} C_DIS
LIN {X 155.771,Y 91.552,Z 45.051,A 180.000,B 0.000,C 180.000} C_DIS
LIN {X 155.771,Y 92.177,Z 45.051,A 180.000,B 0.000,C 180.000} C_DIS
LIN {X 155.230,Y 92.489,Z 45.051,A 180.000,B 0.000,C 180.000} C_DIS
LIN {X 155.120,Y 92.489,Z 45.026,A 180.000,B 0.000,C 180.000} C_DIS
LIN {X 155.010,Y 92.489,Z 45.000,A 180.000,B 0.000,C 180.000} C_DIS
; Cutting Move Starts
LIN {X 152.500,Y 92.489,Z 45.000,A 180.000,B 0.000,C 180.000} C_DIS
LIN {X 152.500,Y 92.489,Z 52.000,A 180.000,B 0.000,C 180.000} C_DIS
LIN {X 150.982,Y 92.489,Z 52.000,A 180.000,B 0.000,C 180.000} C_DIS
LIN {X 150.982,Y 92.489,Z 57.000,A 180.000,B 0.000,C 180.000} C_DIS
LIN {X 131.046,Y 92.489,Z 57.000,A 180.000,B 0.000,C 180.000} C_DIS
LIN {X 131.046,Y 92.489,Z 62.000,A 180.000,B 0.000,C 180.000} C_DIS
LIN {X 111.638,Y 92.489,Z 62.000,A 180.000,B 0.000,C 180.000} C_DIS
LIN {X 111.634,Y 92.489,Z 67.562,A 180.000,B 0.000,C 180.000} C_DIS
LIN {X 109.467,Y 92.489,Z 71.899,A 180.000,B 0.000,C 180.000} C_DIS
LIN {X 107.832,Y 92.489,Z 75.096,A 180.000,B 0.000,C 180.000} C_DIS
LIN {X 106.593,Y 92.489,Z 77.452,A 180.000,B 0.000,C 180.000} C_DIS
LIN {X 105.815,Y 92.489,Z 78.897,A 180.000,B 0.000,C 180.000} C_DIS
LIN {X 105.306,Y 92.489,Z 79.829,A 180.000,B 0.000,C 180.000} C_DIS
LIN {X 104.618,Y 92.489,Z 81.051,A 180.000,B 0.000,C 180.000} C_DIS
LIN {X 103.785,Y 92.489,Z 82.485,A 180.000,B 0.000,C 180.000} C_DIS
LIN {X 103.201,Y 92.489,Z 83.443,A 180.000,B 0.000,C 180.000} C_DIS
LIN {X 102.387,Y 92.489,Z 84.711,A 180.000,B 0.000,C 180.000} C_DIS
LIN {X 101.992,Y 92.489,Z 85.289,A 180.000,B 0.000,C 180.000} C_DIS
LIN {X 101.329,Y 92.489,Z 86.196,A 180.000,B 0.000,C 180.000} C_DIS
LIN {X 101.028,Y 92.489,Z 86.579,A 180.000,B 0.000,C 180.000} C_DIS
LIN {X 100.680,Y 92.489,Z 86.986,A 180.000,B 0.000,C 180.000} C_DIS
LIN {X 100.362,Y 92.489,Z 87.346,A 180.000,B 0.000,C 180.000} C_DIS
LIN {X 100.116,Y 92.489,Z 87.599,A 180.000,B 0.000,C 180.000} C_DIS
LIN {X 99.599,Y 92.489,Z 88.070,A 180.000,B 0.000,C 180.000} C_DIS
LIN {X 99.394,Y 92.489,Z 88.234,A 180.000,B 0.000,C 180.000} C_DIS
LIN {X 99.078,Y 92.489,Z 88.446,A 180.000,B 0.000,C 180.000} C_DIS
LIN {X 98.853,Y 92.489,Z 88.591,A 180.000,B 0.000,C 180.000} C_DIS
LIN {X 98.684,Y 92.489,Z 88.679,A 180.000,B 0.000,C 180.000} C_DIS
LIN {X 98.223,Y 92.489,Z 88.864,A 180.000,B 0.000,C 180.000} C_DIS
LIN {X 98.037,Y 92.489,Z 88.913,A 180.000,B 0.000,C 180.000} C_DIS
LIN {X 97.594,Y 92.489,Z 88.973,A 180.000,B 0.000,C 180.000} C_DIS
LIN {X 97.399,Y 92.489,Z 88.973,A 180.000,B 0.000,C 180.000} C_DIS
LIN {X 96.960,Y 92.489,Z 88.913,A 180.000,B 0.000,C 180.000} C_DIS
LIN {X 96.770,Y 92.489,Z 88.862,A 180.000,B 0.000,C 180.000} C_DIS
LIN {X 96.309,Y 92.489,Z 88.676,A 180.000,B 0.000,C 180.000} C_DIS
LIN {X 96.135,Y 92.489,Z 88.584,A 180.000,B 0.000,C 180.000} C_DIS
LIN {X 95.789,Y 92.489,Z 88.358,A 180.000,B 0.000,C 180.000} C_DIS
LIN {X 95.575,Y 92.489,Z 88.211,A 180.000,B 0.000,C 180.000} C_DIS
LIN {X 95.335,Y 92.489,Z 88.012,A 180.000,B 0.000,C 180.000} C_DIS
LIN {X 94.874,Y 92.489,Z 87.589,A 180.000,B 0.000,C 180.000} C_DIS
LIN {X 94.596,Y 92.489,Z 87.300,A 180.000,B 0.000,C 180.000} C_DIS
LIN {X 94.054,Y 92.489,Z 86.678,A 180.000,B 0.000,C 180.000} C_DIS
LIN {X 93.753,Y 92.489,Z 86.303,A 180.000,B 0.000,C 180.000} C_DIS
LIN {X 93.433,Y 92.489,Z 85.874,A 180.000,B 0.000,C 180.000} C_DIS
LIN {X 92.933,Y 92.489,Z 85.182,A 180.000,B 0.000,C 180.000} C_DIS
LIN {X 92.521,Y 92.489,Z 84.572,A 180.000,B 0.000,C 180.000} C_DIS
LIN {X 91.730,Y 92.489,Z 83.333,A 180.000,B 0.000,C 180.000} C_DIS
LIN {X 91.192,Y 92.489,Z 82.445,A 180.000,B 0.000,C 180.000} C_DIS
LIN {X 90.336,Y 92.489,Z 80.971,A 180.000,B 0.000,C 180.000} C_DIS
LIN {X 89.479,Y 92.489,Z 79.441,A 180.000,B 0.000,C 180.000} C_DIS
LIN {X 88.468,Y 92.489,Z 77.567,A 180.000,B 0.000,C 180.000} C_DIS
LIN {X 87.612,Y 92.489,Z 75.943,A 180.000,B 0.000,C 180.000} C_DIS
LIN {X 86.920,Y 92.489,Z 74.616,A 180.000,B 0.000,C 180.000} C_DIS
LIN {X 85.343,Y 92.489,Z 71.522,A 180.000,B 0.000,C 180.000} C_DIS
LIN {X 83.362,Y 92.489,Z 67.555,A 180.000,B 0.000,C 180.000} C_DIS
LIN {X 83.361,Y 92.489,Z 62.000,A 180.000,B 0.000,C 180.000} C_DIS
LIN {X 67.231,Y 92.489,Z 62.000,A 180.000,B 0.000,C 180.000} C_DIS
LIN {X 67.231,Y 92.489,Z 66.500,A 180.000,B 0.000,C 180.000} C_DIS
LIN {X 67.160,Y 92.489,Z 66.500,A 180.000,B 0.000,C 180.000} C_DIS
LIN {X 67.160,Y 92.489,Z 70.000,A 180.000,B 0.000,C 180.000} C_DIS
LIN {X 49.840,Y 92.489,Z 70.000,A 180.000,B 0.000,C 180.000} C_DIS
LIN {X 49.840,Y 92.489,Z 66.500,A 180.000,B 0.000,C 180.000} C_DIS
LIN {X 49.769,Y 92.489,Z 66.500,A 180.000,B 0.000,C 180.000} C_DIS
LIN {X 49.769,Y 92.489,Z 62.000,A 180.000,B 0.000,C 180.000} C_DIS
LIN {X 23.954,Y 92.489,Z 62.000,A 180.000,B 0.000,C 180.000} C_DIS
LIN {X 23.954,Y 92.489,Z 57.000,A 180.000,B 0.000,C 180.000} C_DIS
LIN {X 4.018,Y 92.489,Z 57.000,A 180.000,B 0.000,C 180.000} C_DIS
LIN {X 4.018,Y 92.489,Z 52.000,A 180.000,B 0.000,C 180.000} C_DIS
LIN {X 2.500,Y 92.489,Z 52.000,A 180.000,B 0.000,C 180.000} C_DIS
LIN {X 2.500,Y 92.489,Z 45.000,A 180.000,B 0.000,C 180.000} C_DIS
LIN {X -0.010,Y 92.489,Z 45.000,A 180.000,B 0.000,C 180.000} C_DIS
; Link Move Starts
LIN {X -0.120,Y 92.489,Z 45.026,A 180.000,B 0.000,C 180.000} C_DIS
LIN {X -0.230,Y 92.489,Z 45.051,A 180.000,B 0.000,C 180.000} C_DIS
LIN {X -0.771,Y 92.802,Z 45.051,A 180.000,B 0.000,C 180.000} C_DIS
LIN {X -0.771,Y 93.427,Z 45.051,A 180.000,B 0.000,C 180.000} C_DIS
LIN {X -0.230,Y 93.739,Z 45.051,A 180.000,B 0.000,C 180.000} C_DIS
LIN {X -0.120,Y 93.739,Z 45.026,A 180.000,B 0.000,C 180.000} C_DIS
LIN {X -0.010,Y 93.739,Z 45.000,A 180.000,B 0.000,C 180.000} C_DIS
; Cutting Move Starts
LIN {X 2.500,Y 93.739,Z 45.000,A 180.000,B 0.000,C 180.000} C_DIS
LIN {X 2.500,Y 93.739,Z 52.000,A 180.000,B 0.000,C 180.000} C_DIS
LIN {X 4.280,Y 93.739,Z 52.000,A 180.000,B 0.000,C 180.000} C_DIS
LIN {X 4.284,Y 93.739,Z 57.000,A 180.000,B 0.000,C 180.000} C_DIS
LIN {X 25.204,Y 93.739,Z 57.000,A 180.000,B 0.000,C 180.000} C_DIS
LIN {X 25.204,Y 93.739,Z 62.000,A 180.000,B 0.000,C 180.000} C_DIS
LIN {X 48.643,Y 93.739,Z 62.000,A 180.000,B 0.000,C 180.000} C_DIS
LIN {X 48.643,Y 93.739,Z 66.500,A 180.000,B 0.000,C 180.000} C_DIS
LIN {X 48.703,Y 93.739,Z 66.500,A 180.000,B 0.000,C 180.000} C_DIS
LIN {X 48.707,Y 93.739,Z 70.000,A 180.000,B 0.000,C 180.000} C_DIS
LIN {X 68.292,Y 93.739,Z 70.000,A 180.000,B 0.000,C 180.000} C_DIS
LIN {X 68.294,Y 93.739,Z 66.500,A 180.000,B 0.000,C 180.000} C_DIS
LIN {X 68.353,Y 93.739,Z 66.500,A 180.000,B 0.000,C 180.000} C_DIS
LIN {X 68.357,Y 93.739,Z 62.000,A 180.000,B 0.000,C 180.000} C_DIS
LIN {X 82.984,Y 93.739,Z 62.000,A 180.000,B 0.000,C 180.000} C_DIS
LIN {X 82.984,Y 93.739,Z 67.555,A 180.000,B 0.000,C 180.000} C_DIS
LIN {X 84.259,Y 93.739,Z 70.202,A 180.000,B 0.000,C 180.000} C_DIS
LIN {X 85.571,Y 93.739,Z 72.891,A 180.000,B 0.000,C 180.000} C_DIS
LIN {X 86.853,Y 93.739,Z 75.505,A 180.000,B 0.000,C 180.000} C_DIS
LIN {X 88.605,Y 93.739,Z 79.010,A 180.000,B 0.000,C 180.000} C_DIS
LIN {X 89.754,Y 93.739,Z 81.255,A 180.000,B 0.000,C 180.000} C_DIS
LIN {X 90.625,Y 93.739,Z 82.910,A 180.000,B 0.000,C 180.000} C_DIS
LIN {X 91.358,Y 93.739,Z 84.275,A 180.000,B 0.000,C 180.000} C_DIS
LIN {X 91.855,Y 93.739,Z 85.173,A 180.000,B 0.000,C 180.000} C_DIS
LIN {X 92.479,Y 93.739,Z 86.262,A 180.000,B 0.000,C 180.000} C_DIS
LIN {X 92.923,Y 93.739,Z 87.018,A 180.000,B 0.000,C 180.000} C_DIS
LIN {X 93.298,Y 93.739,Z 87.622,A 180.000,B 0.000,C 180.000} C_DIS
LIN {X 93.893,Y 93.739,Z 88.546,A 180.000,B 0.000,C 180.000} C_DIS
LIN {X 94.209,Y 93.739,Z 88.998,A 180.000,B 0.000,C 180.000} C_DIS
LIN {X 100.789,Y 93.739,Z 89.000,A 180.000,B 0.000,C 180.000} C_DIS
LIN {X 100.801,Y 93.739,Z 88.985,A 180.000,B 0.000,C 180.000} C_DIS
LIN {X 101.110,Y 93.739,Z 88.543,A 180.000,B 0.000,C 180.000} C_DIS
LIN {X 101.725,Y 93.739,Z 87.586,A 180.000,B 0.000,C 180.000} C_DIS
LIN {X 102.088,Y 93.739,Z 87.000,A 180.000,B 0.000,C 180.000} C_DIS
LIN {X 102.551,Y 93.739,Z 86.209,A 180.000,B 0.000,C 180.000} C_DIS
LIN {X 103.151,Y 93.739,Z 85.162,A 180.000,B 0.000,C 180.000} C_DIS
LIN {X 103.649,Y 93.739,Z 84.263,A 180.000,B 0.000,C 180.000} C_DIS
LIN {X 104.379,Y 93.739,Z 82.902,A 180.000,B 0.000,C 180.000} C_DIS
LIN {X 105.250,Y 93.739,Z 81.249,A 180.000,B 0.000,C 180.000} C_DIS
LIN {X 106.404,Y 93.739,Z 78.992,A 180.000,B 0.000,C 180.000} C_DIS
LIN {X 108.179,Y 93.739,Z 75.442,A 180.000,B 0.000,C 180.000} C_DIS
LIN {X 110.313,Y 93.739,Z 71.084,A 180.000,B 0.000,C 180.000} C_DIS
LIN {X 112.014,Y 93.739,Z 67.559,A 180.000,B 0.000,C 180.000} C_DIS
LIN {X 112.016,Y 93.739,Z 62.000,A 180.000,B 0.000,C 180.000} C_DIS
LIN {X 129.795,Y 93.739,Z 62.000,A 180.000,B 0.000,C 180.000} C_DIS
LIN {X 129.796,Y 93.739,Z 57.000,A 180.000,B 0.000,C 180.000} C_DIS
LIN {X 150.716,Y 93.739,Z 57.000,A 180.000,B 0.000,C 180.000} C_DIS
LIN {X 150.716,Y 93.739,Z 52.000,A 180.000,B 0.000,C 180.000} C_DIS
LIN {X 152.500,Y 93.739,Z 52.000,A 180.000,B 0.000,C 180.000} C_DIS
LIN {X 152.500,Y 93.739,Z 45.000,A 180.000,B 0.000,C 180.000} C_DIS
LIN {X 155.010,Y 93.739,Z 45.000,A 180.000,B 0.000,C 180.000} C_DIS
; Link Move Starts
LIN {X 155.120,Y 93.739,Z 45.026,A 180.000,B 0.000,C 180.000} C_DIS
LIN {X 155.230,Y 93.739,Z 45.051,A 180.000,B 0.000,C 180.000} C_DIS
LIN {X 155.771,Y 94.052,Z 45.051,A 180.000,B 0.000,C 180.000} C_DIS
LIN {X 155.771,Y 94.677,Z 45.051,A 180.000,B 0.000,C 180.000} C_DIS
LIN {X 155.230,Y 94.989,Z 45.051,A 180.000,B 0.000,C 180.000} C_DIS
LIN {X 155.120,Y 94.989,Z 45.026,A 180.000,B 0.000,C 180.000} C_DIS
LIN {X 155.010,Y 94.989,Z 45.000,A 180.000,B 0.000,C 180.000} C_DIS
; Cutting Move Starts
LIN {X 152.500,Y 94.989,Z 45.000,A 180.000,B 0.000,C 180.000} C_DIS
LIN {X 152.500,Y 94.989,Z 52.000,A 180.000,B 0.000,C 180.000} C_DIS
LIN {X 150.432,Y 94.989,Z 52.000,A 180.000,B 0.000,C 180.000} C_DIS
LIN {X 150.432,Y 94.989,Z 57.000,A 180.000,B 0.000,C 180.000} C_DIS
LIN {X 128.546,Y 94.989,Z 57.000,A 180.000,B 0.000,C 180.000} C_DIS
LIN {X 128.546,Y 94.989,Z 62.000,A 180.000,B 0.000,C 180.000} C_DIS
LIN {X 112.288,Y 94.989,Z 62.000,A 180.000,B 0.000,C 180.000} C_DIS
LIN {X 112.287,Y 94.989,Z 67.559,A 180.000,B 0.000,C 180.000} C_DIS
LIN {X 108.474,Y 94.989,Z 75.579,A 180.000,B 0.000,C 180.000} C_DIS
LIN {X 105.869,Y 94.989,Z 80.982,A 180.000,B 0.000,C 180.000} C_DIS
LIN {X 104.642,Y 94.989,Z 83.486,A 180.000,B 0.000,C 180.000} C_DIS
LIN {X 103.185,Y 94.989,Z 86.393,A 180.000,B 0.000,C 180.000} C_DIS
LIN {X 102.571,Y 94.989,Z 87.585,A 180.000,B 0.000,C 180.000} C_DIS
LIN {X 101.819,Y 94.989,Z 89.000,A 180.000,B 0.000,C 180.000} C_DIS
LIN {X 93.180,Y 94.989,Z 88.999,A 180.000,B 0.000,C 180.000} C_DIS
LIN {X 92.331,Y 94.989,Z 87.399,A 180.000,B 0.000,C 180.000} C_DIS
LIN {X 91.657,Y 94.989,Z 86.081,A 180.000,B 0.000,C 180.000} C_DIS
LIN {X 90.222,Y 94.989,Z 83.211,A 180.000,B 0.000,C 180.000} C_DIS
LIN {X 88.806,Y 94.989,Z 80.314,A 180.000,B 0.000,C 180.000} C_DIS
LIN {X 86.153,Y 94.989,Z 74.798,A 180.000,B 0.000,C 180.000} C_DIS
LIN {X 82.712,Y 94.989,Z 67.555,A 180.000,B 0.000,C 180.000} C_DIS
LIN {X 82.711,Y 94.989,Z 62.000,A 180.000,B 0.000,C 180.000} C_DIS
LIN {X 69.224,Y 94.989,Z 62.000,A 180.000,B 0.000,C 180.000} C_DIS
LIN {X 69.224,Y 94.989,Z 66.500,A 180.000,B 0.000,C 180.000} C_DIS
LIN {X 69.166,Y 94.989,Z 66.500,A 180.000,B 0.000,C 180.000} C_DIS
LIN {X 69.164,Y 94.989,Z 70.000,A 180.000,B 0.000,C 180.000} C_DIS
LIN {X 62.316,Y 94.989,Z 70.000,A 180.000,B 0.000,C 180.000} C_DIS
LIN {X 62.316,Y 94.989,Z 74.500,A 180.000,B 0.000,C 180.000} C_DIS
LIN {X 62.213,Y 94.989,Z 74.500,A 180.000,B 0.000,C 180.000} C_DIS
LIN {X 62.213,Y 94.989,Z 78.000,A 180.000,B 0.000,C 180.000} C_DIS
LIN {X 54.779,Y 94.989,Z 78.000,A 180.000,B 0.000,C 180.000} C_DIS
LIN {X 54.779,Y 94.989,Z 74.500,A 180.000,B 0.000,C 180.000} C_DIS
LIN {X 54.684,Y 94.989,Z 74.500,A 180.000,B 0.000,C 180.000} C_DIS
LIN {X 54.683,Y 94.989,Z 70.000,A 180.000,B 0.000,C 180.000} C_DIS
LIN {X 47.834,Y 94.989,Z 70.000,A 180.000,B 0.000,C 180.000} C_DIS
LIN {X 47.834,Y 94.989,Z 66.500,A 180.000,B 0.000,C 180.000} C_DIS
LIN {X 47.776,Y 94.989,Z 66.500,A 180.000,B 0.000,C 180.000} C_DIS
LIN {X 47.776,Y 94.989,Z 62.000,A 180.000,B 0.000,C 180.000} C_DIS
LIN {X 26.454,Y 94.989,Z 62.000,A 180.000,B 0.000,C 180.000} C_DIS
LIN {X 26.453,Y 94.989,Z 57.000,A 180.000,B 0.000,C 180.000} C_DIS
LIN {X 4.568,Y 94.989,Z 57.000,A 180.000,B 0.000,C 180.000} C_DIS
LIN {X 4.566,Y 94.989,Z 52.000,A 180.000,B 0.000,C 180.000} C_DIS
LIN {X 2.500,Y 94.989,Z 52.000,A 180.000,B 0.000,C 180.000} C_DIS
LIN {X 2.500,Y 94.989,Z 45.000,A 180.000,B 0.000,C 180.000} C_DIS
LIN {X -0.010,Y 94.989,Z 45.000,A 180.000,B 0.000,C 180.000} C_DIS
; Link Move Starts
LIN {X -0.120,Y 94.989,Z 45.026,A 180.000,B 0.000,C 180.000} C_DIS
LIN {X -0.230,Y 94.989,Z 45.051,A 180.000,B 0.000,C 180.000} C_DIS
LIN {X -0.771,Y 95.302,Z 45.051,A 180.000,B 0.000,C 180.000} C_DIS
LIN {X -0.771,Y 95.926,Z 45.051,A 180.000,B 0.000,C 180.000} C_DIS
LIN {X -0.230,Y 96.239,Z 45.051,A 180.000,B 0.000,C 180.000} C_DIS
LIN {X -0.120,Y 96.239,Z 45.026,A 180.000,B 0.000,C 180.000} C_DIS
LIN {X -0.010,Y 96.239,Z 45.000,A 180.000,B 0.000,C 180.000} C_DIS
; Cutting Move Starts
LIN {X 2.500,Y 96.239,Z 45.000,A 180.000,B 0.000,C 180.000} C_DIS
LIN {X 2.500,Y 96.239,Z 52.000,A 180.000,B 0.000,C 180.000} C_DIS
LIN {X 4.882,Y 96.239,Z 52.000,A 180.000,B 0.000,C 180.000} C_DIS
LIN {X 4.882,Y 96.239,Z 57.000,A 180.000,B 0.000,C 180.000} C_DIS
LIN {X 27.701,Y 96.239,Z 57.000,A 180.000,B 0.000,C 180.000} C_DIS
LIN {X 27.703,Y 96.239,Z 62.000,A 180.000,B 0.000,C 180.000} C_DIS
LIN {X 47.103,Y 96.239,Z 62.000,A 180.000,B 0.000,C 180.000} C_DIS
LIN {X 47.107,Y 96.239,Z 66.500,A 180.000,B 0.000,C 180.000} C_DIS
LIN {X 47.162,Y 96.239,Z 66.500,A 180.000,B 0.000,C 180.000} C_DIS
LIN {X 47.162,Y 96.239,Z 70.000,A 180.000,B 0.000,C 180.000} C_DIS
LIN {X 53.090,Y 96.239,Z 70.000,A 180.000,B 0.000,C 180.000} C_DIS
LIN {X 53.090,Y 96.239,Z 74.500,A 180.000,B 0.000,C 180.000} C_DIS
LIN {X 53.157,Y 96.239,Z 74.500,A 180.000,B 0.000,C 180.000} C_DIS
LIN {X 53.158,Y 96.239,Z 78.000,A 180.000,B 0.000,C 180.000} C_DIS
LIN {X 63.839,Y 96.239,Z 78.000,A 180.000,B 0.000,C 180.000} C_DIS
LIN {X 63.840,Y 96.239,Z 74.500,A 180.000,B 0.000,C 180.000} C_DIS
LIN {X 63.912,Y 96.239,Z 74.500,A 180.000,B 0.000,C 180.000} C_DIS
LIN {X 63.912,Y 96.239,Z 70.000,A 180.000,B 0.000,C 180.000} C_DIS
LIN {X 69.837,Y 96.239,Z 70.000,A 180.000,B 0.000,C 180.000} C_DIS
LIN {X 69.838,Y 96.239,Z 66.500,A 180.000,B 0.000,C 180.000} C_DIS
LIN {X 69.893,Y 96.239,Z 66.500,A 180.000,B 0.000,C 180.000} C_DIS
LIN {X 69.893,Y 96.239,Z 62.000,A 180.000,B 0.000,C 180.000} C_DIS
LIN {X 82.558,Y 96.239,Z 62.000,A 180.000,B 0.000,C 180.000} C_DIS
LIN {X 82.558,Y 96.239,Z 67.555,A 180.000,B 0.000,C 180.000} C_DIS
LIN {X 85.410,Y 96.239,Z 73.653,A 180.000,B 0.000,C 180.000} C_DIS
LIN {X 89.515,Y 96.239,Z 82.381,A 180.000,B 0.000,C 180.000} C_DIS
LIN {X 91.293,Y 96.239,Z 86.139,A 180.000,B 0.000,C 180.000} C_DIS
LIN {X 92.666,Y 96.239,Z 88.999,A 180.000,B 0.000,C 180.000} C_DIS
LIN {X 102.332,Y 96.239,Z 89.000,A 180.000,B 0.000,C 180.000} C_DIS
LIN {X 103.092,Y 96.239,Z 87.423,A 180.000,B 0.000,C 180.000} C_DIS
LIN {X 104.454,Y 96.239,Z 84.567,A 180.000,B 0.000,C 180.000} C_DIS
LIN {X 108.613,Y 96.239,Z 75.734,A 180.000,B 0.000,C 180.000} C_DIS
LIN {X 112.442,Y 96.239,Z 67.555,A 180.000,B 0.000,C 180.000} C_DIS
LIN {X 112.442,Y 96.239,Z 62.000,A 180.000,B 0.000,C 180.000} C_DIS
LIN {X 127.297,Y 96.239,Z 62.000,A 180.000,B 0.000,C 180.000} C_DIS
LIN {X 127.297,Y 96.239,Z 57.000,A 180.000,B 0.000,C 180.000} C_DIS
LIN {X 150.118,Y 96.239,Z 57.000,A 180.000,B 0.000,C 180.000} C_DIS
LIN {X 150.118,Y 96.239,Z 52.000,A 180.000,B 0.000,C 180.000} C_DIS
LIN {X 152.500,Y 96.239,Z 52.000,A 180.000,B 0.000,C 180.000} C_DIS
LIN {X 152.500,Y 96.239,Z 45.000,A 180.000,B 0.000,C 180.000} C_DIS
LIN {X 155.010,Y 96.239,Z 45.000,A 180.000,B 0.000,C 180.000} C_DIS
; Link Move Starts
LIN {X 155.120,Y 96.239,Z 45.026,A 180.000,B 0.000,C 180.000} C_DIS
LIN {X 155.230,Y 96.239,Z 45.051,A 180.000,B 0.000,C 180.000} C_DIS
LIN {X 155.771,Y 96.551,Z 45.051,A 180.000,B 0.000,C 180.000} C_DIS
LIN {X 155.771,Y 97.176,Z 45.051,A 180.000,B 0.000,C 180.000} C_DIS
LIN {X 155.230,Y 97.489,Z 45.051,A 180.000,B 0.000,C 180.000} C_DIS
LIN {X 155.120,Y 97.489,Z 45.026,A 180.000,B 0.000,C 180.000} C_DIS
LIN {X 155.010,Y 97.489,Z 45.000,A 180.000,B 0.000,C 180.000} C_DIS
; Cutting Move Starts
LIN {X 152.500,Y 97.489,Z 45.000,A 180.000,B 0.000,C 180.000} C_DIS
LIN {X 152.500,Y 97.489,Z 52.000,A 180.000,B 0.000,C 180.000} C_DIS
LIN {X 149.782,Y 97.489,Z 52.000,A 180.000,B 0.000,C 180.000} C_DIS
LIN {X 149.782,Y 97.489,Z 57.000,A 180.000,B 0.000,C 180.000} C_DIS
LIN {X 126.047,Y 97.489,Z 57.000,A 180.000,B 0.000,C 180.000} C_DIS
LIN {X 126.044,Y 97.489,Z 62.000,A 180.000,B 0.000,C 180.000} C_DIS
LIN {X 112.500,Y 97.489,Z 62.000,A 180.000,B 0.000,C 180.000} C_DIS
LIN {X 112.497,Y 97.489,Z 67.562,A 180.000,B 0.000,C 180.000} C_DIS
LIN {X 102.495,Y 97.489,Z 89.000,A 180.000,B 0.000,C 180.000} C_DIS
LIN {X 92.505,Y 97.489,Z 89.000,A 180.000,B 0.000,C 180.000} C_DIS
LIN {X 82.500,Y 97.489,Z 67.555,A 180.000,B 0.000,C 180.000} C_DIS
LIN {X 82.500,Y 97.489,Z 62.000,A 180.000,B 0.000,C 180.000} C_DIS
LIN {X 70.389,Y 97.489,Z 62.000,A 180.000,B 0.000,C 180.000} C_DIS
LIN {X 70.389,Y 97.489,Z 66.500,A 180.000,B 0.000,C 180.000} C_DIS
LIN {X 70.336,Y 97.489,Z 66.500,A 180.000,B 0.000,C 180.000} C_DIS
LIN {X 70.333,Y 97.489,Z 70.000,A 180.000,B 0.000,C 180.000} C_DIS
LIN {X 64.894,Y 97.489,Z 70.000,A 180.000,B 0.000,C 180.000} C_DIS
LIN {X 64.893,Y 97.489,Z 74.500,A 180.000,B 0.000,C 180.000} C_DIS
LIN {X 64.836,Y 97.489,Z 74.500,A 180.000,B 0.000,C 180.000} C_DIS
LIN {X 64.836,Y 97.489,Z 78.000,A 180.000,B 0.000,C 180.000} C_DIS
LIN {X 52.168,Y 97.489,Z 78.000,A 180.000,B 0.000,C 180.000} C_DIS
LIN {X 52.168,Y 97.489,Z 74.500,A 180.000,B 0.000,C 180.000} C_DIS
LIN {X 52.109,Y 97.489,Z 74.500,A 180.000,B 0.000,C 180.000} C_DIS
LIN {X 52.109,Y 97.489,Z 70.000,A 180.000,B 0.000,C 180.000} C_DIS
LIN {X 46.664,Y 97.489,Z 70.000,A 180.000,B 0.000,C 180.000} C_DIS
LIN {X 46.664,Y 97.489,Z 66.500,A 180.000,B 0.000,C 180.000} C_DIS
LIN {X 46.611,Y 97.489,Z 66.500,A 180.000,B 0.000,C 180.000} C_DIS
LIN {X 46.611,Y 97.489,Z 62.000,A 180.000,B 0.000,C 180.000} C_DIS
LIN {X 28.953,Y 97.489,Z 62.000,A 180.000,B 0.000,C 180.000} C_DIS
LIN {X 28.953,Y 97.489,Z 57.000,A 180.000,B 0.000,C 180.000} C_DIS
LIN {X 5.218,Y 97.489,Z 57.000,A 180.000,B 0.000,C 180.000} C_DIS
LIN {X 5.214,Y 97.489,Z 52.000,A 180.000,B 0.000,C 180.000} C_DIS
LIN {X 2.500,Y 97.489,Z 52.000,A 180.000,B 0.000,C 180.000} C_DIS
LIN {X 2.500,Y 97.489,Z 45.000,A 180.000,B 0.000,C 180.000} C_DIS
LIN {X -0.010,Y 97.489,Z 45.000,A 180.000,B 0.000,C 180.000} C_DIS
; Link Move Starts
LIN {X -0.120,Y 97.489,Z 45.026,A 180.000,B 0.000,C 180.000} C_DIS
LIN {X -0.230,Y 97.489,Z 45.051,A 180.000,B 0.000,C 180.000} C_DIS
LIN {X -0.771,Y 97.801,Z 45.051,A 180.000,B 0.000,C 180.000} C_DIS
LIN {X -0.771,Y 98.426,Z 45.051,A 180.000,B 0.000,C 180.000} C_DIS
LIN {X -0.230,Y 98.739,Z 45.051,A 180.000,B 0.000,C 180.000} C_DIS
LIN {X -0.120,Y 98.739,Z 45.026,A 180.000,B 0.000,C 180.000} C_DIS
LIN {X -0.010,Y 98.739,Z 45.000,A 180.000,B 0.000,C 180.000} C_DIS
; Cutting Move Starts
LIN {X 2.500,Y 98.739,Z 45.000,A 180.000,B 0.000,C 180.000} C_DIS
LIN {X 2.500,Y 98.739,Z 52.000,A 180.000,B 0.000,C 180.000} C_DIS
LIN {X 5.574,Y 98.739,Z 52.000,A 180.000,B 0.000,C 180.000} C_DIS
LIN {X 5.574,Y 98.739,Z 57.000,A 180.000,B 0.000,C 180.000} C_DIS
LIN {X 30.203,Y 98.739,Z 57.000,A 180.000,B 0.000,C 180.000} C_DIS
LIN {X 30.203,Y 98.739,Z 62.000,A 180.000,B 0.000,C 180.000} C_DIS
LIN {X 46.263,Y 98.739,Z 62.000,A 180.000,B 0.000,C 180.000} C_DIS
LIN {X 46.263,Y 98.739,Z 66.500,A 180.000,B 0.000,C 180.000} C_DIS
LIN {X 46.314,Y 98.739,Z 66.500,A 180.000,B 0.000,C 180.000} C_DIS
LIN {X 46.314,Y 98.739,Z 70.000,A 180.000,B 0.000,C 180.000} C_DIS
LIN {X 51.476,Y 98.739,Z 70.000,A 180.000,B 0.000,C 180.000} C_DIS
LIN {X 51.476,Y 98.739,Z 74.500,A 180.000,B 0.000,C 180.000} C_DIS
LIN {X 51.530,Y 98.739,Z 74.500,A 180.000,B 0.000,C 180.000} C_DIS
LIN {X 51.530,Y 98.739,Z 78.000,A 180.000,B 0.000,C 180.000} C_DIS
LIN {X 65.467,Y 98.739,Z 78.000,A 180.000,B 0.000,C 180.000} C_DIS
LIN {X 65.470,Y 98.739,Z 74.500,A 180.000,B 0.000,C 180.000} C_DIS
LIN {X 65.523,Y 98.739,Z 74.500,A 180.000,B 0.000,C 180.000} C_DIS
LIN {X 65.523,Y 98.739,Z 70.000,A 180.000,B 0.000,C 180.000} C_DIS
LIN {X 70.686,Y 98.739,Z 70.000,A 180.000,B 0.000,C 180.000} C_DIS
LIN {X 70.686,Y 98.739,Z 66.500,A 180.000,B 0.000,C 180.000} C_DIS
LIN {X 70.737,Y 98.739,Z 66.500,A 180.000,B 0.000,C 180.000} C_DIS
LIN {X 70.737,Y 98.739,Z 62.000,A 180.000,B 0.000,C 180.000} C_DIS
LIN {X 82.554,Y 98.739,Z 62.000,A 180.000,B 0.000,C 180.000} C_DIS
LIN {X 82.556,Y 98.739,Z 67.555,A 180.000,B 0.000,C 180.000} C_DIS
LIN {X 85.530,Y 98.739,Z 73.913,A 180.000,B 0.000,C 180.000} C_DIS
LIN {X 89.513,Y 98.739,Z 82.383,A 180.000,B 0.000,C 180.000} C_DIS
LIN {X 91.359,Y 98.739,Z 86.287,A 180.000,B 0.000,C 180.000} C_DIS
LIN {X 92.660,Y 98.739,Z 88.999,A 180.000,B 0.000,C 180.000} C_DIS
LIN {X 102.338,Y 98.739,Z 89.000,A 180.000,B 0.000,C 180.000} C_DIS
LIN {X 102.994,Y 98.739,Z 87.640,A 180.000,B 0.000,C 180.000} C_DIS
LIN {X 104.321,Y 98.739,Z 84.855,A 180.000,B 0.000,C 180.000} C_DIS
LIN {X 108.446,Y 98.739,Z 76.094,A 180.000,B 0.000,C 180.000} C_DIS
LIN {X 112.444,Y 98.739,Z 67.555,A 180.000,B 0.000,C 180.000} C_DIS
LIN {X 112.444,Y 98.739,Z 62.000,A 180.000,B 0.000,C 180.000} C_DIS
LIN {X 124.797,Y 98.739,Z 62.000,A 180.000,B 0.000,C 180.000} C_DIS
LIN {X 124.797,Y 98.739,Z 57.000,A 180.000,B 0.000,C 180.000} C_DIS
LIN {X 149.424,Y 98.739,Z 57.000,A 180.000,B 0.000,C 180.000} C_DIS
LIN {X 149.426,Y 98.739,Z 52.000,A 180.000,B 0.000,C 180.000} C_DIS
LIN {X 152.500,Y 98.739,Z 52.000,A 180.000,B 0.000,C 180.000} C_DIS
LIN {X 152.500,Y 98.739,Z 45.000,A 180.000,B 0.000,C 180.000} C_DIS
LIN {X 155.010,Y 98.739,Z 45.000,A 180.000,B 0.000,C 180.000} C_DIS
; Link Move Starts
LIN {X 155.120,Y 98.739,Z 45.026,A 180.000,B 0.000,C 180.000} C_DIS
LIN {X 155.230,Y 98.739,Z 45.051,A 180.000,B 0.000,C 180.000} C_DIS
LIN {X 155.771,Y 99.051,Z 45.051,A 180.000,B 0.000,C 180.000} C_DIS
LIN {X 155.771,Y 99.676,Z 45.051,A 180.000,B 0.000,C 180.000} C_DIS
LIN {X 155.230,Y 99.989,Z 45.051,A 180.000,B 0.000,C 180.000} C_DIS
LIN {X 155.120,Y 99.989,Z 45.026,A 180.000,B 0.000,C 180.000} C_DIS
LIN {X 155.010,Y 99.989,Z 45.000,A 180.000,B 0.000,C 180.000} C_DIS
; Cutting Move Starts
LIN {X 152.500,Y 99.989,Z 45.000,A 180.000,B 0.000,C 180.000} C_DIS
LIN {X 152.500,Y 99.989,Z 52.000,A 180.000,B 0.000,C 180.000} C_DIS
LIN {X 149.049,Y 99.989,Z 52.000,A 180.000,B 0.000,C 180.000} C_DIS
LIN {X 149.049,Y 99.989,Z 57.000,A 180.000,B 0.000,C 180.000} C_DIS
LIN {X 123.547,Y 99.989,Z 57.000,A 180.000,B 0.000,C 180.000} C_DIS
LIN {X 123.547,Y 99.989,Z 62.000,A 180.000,B 0.000,C 180.000} C_DIS
LIN {X 112.292,Y 99.989,Z 62.000,A 180.000,B 0.000,C 180.000} C_DIS
LIN {X 112.288,Y 99.989,Z 67.562,A 180.000,B 0.000,C 180.000} C_DIS
LIN {X 108.391,Y 99.989,Z 75.762,A 180.000,B 0.000,C 180.000} C_DIS
LIN {X 105.790,Y 99.989,Z 81.159,A 180.000,B 0.000,C 180.000} C_DIS
LIN {X 104.577,Y 99.989,Z 83.633,A 180.000,B 0.000,C 180.000} C_DIS
LIN {X 103.122,Y 99.989,Z 86.536,A 180.000,B 0.000,C 180.000} C_DIS
LIN {X 102.510,Y 99.989,Z 87.724,A 180.000,B 0.000,C 180.000} C_DIS
LIN {X 101.831,Y 99.989,Z 89.000,A 180.000,B 0.000,C 180.000} C_DIS
LIN {X 93.167,Y 99.989,Z 88.999,A 180.000,B 0.000,C 180.000} C_DIS
LIN {X 92.364,Y 99.989,Z 87.483,A 180.000,B 0.000,C 180.000} C_DIS
LIN {X 91.684,Y 99.989,Z 86.151,A 180.000,B 0.000,C 180.000} C_DIS
LIN {X 90.271,Y 99.989,Z 83.327,A 180.000,B 0.000,C 180.000} C_DIS
LIN {X 88.879,Y 99.989,Z 80.478,A 180.000,B 0.000,C 180.000} C_DIS
LIN {X 86.245,Y 99.989,Z 75.002,A 180.000,B 0.000,C 180.000} C_DIS
LIN {X 82.708,Y 99.989,Z 67.555,A 180.000,B 0.000,C 180.000} C_DIS
LIN {X 82.707,Y 99.989,Z 62.000,A 180.000,B 0.000,C 180.000} C_DIS
LIN {X 70.958,Y 99.989,Z 62.000,A 180.000,B 0.000,C 180.000} C_DIS
LIN {X 70.958,Y 99.989,Z 66.500,A 180.000,B 0.000,C 180.000} C_DIS
LIN {X 70.908,Y 99.989,Z 66.500,A 180.000,B 0.000,C 180.000} C_DIS
LIN {X 70.906,Y 99.989,Z 70.000,A 180.000,B 0.000,C 180.000} C_DIS
LIN {X 65.894,Y 99.989,Z 70.000,A 180.000,B 0.000,C 180.000} C_DIS
LIN {X 65.894,Y 99.989,Z 74.500,A 180.000,B 0.000,C 180.000} C_DIS
LIN {X 65.844,Y 99.989,Z 74.500,A 180.000,B 0.000,C 180.000} C_DIS
LIN {X 65.842,Y 99.989,Z 78.000,A 180.000,B 0.000,C 180.000} C_DIS
LIN {X 51.158,Y 99.989,Z 78.000,A 180.000,B 0.000,C 180.000} C_DIS
LIN {X 51.158,Y 99.989,Z 74.500,A 180.000,B 0.000,C 180.000} C_DIS
LIN {X 51.106,Y 99.989,Z 74.500,A 180.000,B 0.000,C 180.000} C_DIS
LIN {X 51.106,Y 99.989,Z 70.000,A 180.000,B 0.000,C 180.000} C_DIS
LIN {X 46.092,Y 99.989,Z 70.000,A 180.000,B 0.000,C 180.000} C_DIS
LIN {X 46.092,Y 99.989,Z 66.500,A 180.000,B 0.000,C 180.000} C_DIS
LIN {X 46.042,Y 99.989,Z 66.500,A 180.000,B 0.000,C 180.000} C_DIS
LIN {X 46.041,Y 99.989,Z 62.000,A 180.000,B 0.000,C 180.000} C_DIS
LIN {X 31.453,Y 99.989,Z 62.000,A 180.000,B 0.000,C 180.000} C_DIS
LIN {X 31.453,Y 99.989,Z 57.000,A 180.000,B 0.000,C 180.000} C_DIS
LIN {X 5.951,Y 99.989,Z 57.000,A 180.000,B 0.000,C 180.000} C_DIS
LIN {X 5.951,Y 99.989,Z 52.000,A 180.000,B 0.000,C 180.000} C_DIS
LIN {X 2.500,Y 99.989,Z 52.000,A 180.000,B 0.000,C 180.000} C_DIS
LIN {X 2.500,Y 99.989,Z 45.000,A 180.000,B 0.000,C 180.000} C_DIS
LIN {X -0.010,Y 99.989,Z 45.000,A 180.000,B 0.000,C 180.000} C_DIS
; Link Move Starts
LIN {X -0.120,Y 99.989,Z 45.026,A 180.000,B 0.000,C 180.000} C_DIS
LIN {X -0.230,Y 99.989,Z 45.051,A 180.000,B 0.000,C 180.000} C_DIS
LIN {X -0.771,Y 100.301,Z 45.051,A 180.000,B 0.000,C 180.000} C_DIS
LIN {X -0.771,Y 100.926,Z 45.051,A 180.000,B 0.000,C 180.000} C_DIS
LIN {X -0.230,Y 101.239,Z 45.051,A 180.000,B 0.000,C 180.000} C_DIS
LIN {X -0.120,Y 101.239,Z 45.026,A 180.000,B 0.000,C 180.000} C_DIS
LIN {X -0.010,Y 101.239,Z 45.000,A 180.000,B 0.000,C 180.000} C_DIS
; Cutting Move Starts
LIN {X 2.500,Y 101.239,Z 45.000,A 180.000,B 0.000,C 180.000} C_DIS
LIN {X 2.500,Y 101.239,Z 52.000,A 180.000,B 0.000,C 180.000} C_DIS
LIN {X 6.360,Y 101.239,Z 52.000,A 180.000,B 0.000,C 180.000} C_DIS
LIN {X 6.360,Y 101.239,Z 57.000,A 180.000,B 0.000,C 180.000} C_DIS
LIN {X 32.701,Y 101.239,Z 57.000,A 180.000,B 0.000,C 180.000} C_DIS
LIN {X 32.703,Y 101.239,Z 62.000,A 180.000,B 0.000,C 180.000} C_DIS
LIN {X 45.957,Y 101.239,Z 62.000,A 180.000,B 0.000,C 180.000} C_DIS
LIN {X 45.957,Y 101.239,Z 66.500,A 180.000,B 0.000,C 180.000} C_DIS
LIN {X 46.007,Y 101.239,Z 66.500,A 180.000,B 0.000,C 180.000} C_DIS
LIN {X 46.007,Y 101.239,Z 70.000,A 180.000,B 0.000,C 180.000} C_DIS
LIN {X 50.959,Y 101.239,Z 70.000,A 180.000,B 0.000,C 180.000} C_DIS
LIN {X 50.959,Y 101.239,Z 74.500,A 180.000,B 0.000,C 180.000} C_DIS
LIN {X 51.009,Y 101.239,Z 74.500,A 180.000,B 0.000,C 180.000} C_DIS
LIN {X 51.009,Y 101.239,Z 78.000,A 180.000,B 0.000,C 180.000} C_DIS
LIN {X 65.995,Y 101.239,Z 78.000,A 180.000,B 0.000,C 180.000} C_DIS
LIN {X 65.995,Y 101.239,Z 74.500,A 180.000,B 0.000,C 180.000} C_DIS
LIN {X 66.045,Y 101.239,Z 74.500,A 180.000,B 0.000,C 180.000} C_DIS
LIN {X 66.045,Y 101.239,Z 70.000,A 180.000,B 0.000,C 180.000} C_DIS
LIN {X 70.993,Y 101.239,Z 70.000,A 180.000,B 0.000,C 180.000} C_DIS
LIN {X 70.993,Y 101.239,Z 66.500,A 180.000,B 0.000,C 180.000} C_DIS
LIN {X 71.041,Y 101.239,Z 66.500,A 180.000,B 0.000,C 180.000} C_DIS
LIN {X 71.043,Y 101.239,Z 62.000,A 180.000,B 0.000,C 180.000} C_DIS
LIN {X 82.978,Y 101.239,Z 62.000,A 180.000,B 0.000,C 180.000} C_DIS
LIN {X 82.978,Y 101.239,Z 67.555,A 180.000,B 0.000,C 180.000} C_DIS
LIN {X 84.401,Y 101.239,Z 70.509,A 180.000,B 0.000,C 180.000} C_DIS
LIN {X 86.631,Y 101.239,Z 75.073,A 180.000,B 0.000,C 180.000} C_DIS
LIN {X 88.247,Y 101.239,Z 78.314,A 180.000,B 0.000,C 180.000} C_DIS
LIN {X 89.053,Y 101.239,Z 79.909,A 180.000,B 0.000,C 180.000} C_DIS
LIN {X 89.843,Y 101.239,Z 81.448,A 180.000,B 0.000,C 180.000} C_DIS
LIN {X 90.685,Y 101.239,Z 83.046,A 180.000,B 0.000,C 180.000} C_DIS
LIN {X 91.414,Y 101.239,Z 84.403,A 180.000,B 0.000,C 180.000} C_DIS
LIN {X 91.918,Y 101.239,Z 85.312,A 180.000,B 0.000,C 180.000} C_DIS
LIN {X 92.728,Y 101.239,Z 86.718,A 180.000,B 0.000,C 180.000} C_DIS
LIN {X 93.125,Y 101.239,Z 87.380,A 180.000,B 0.000,C 180.000} C_DIS
LIN {X 93.840,Y 101.239,Z 88.501,A 180.000,B 0.000,C 180.000} C_DIS
LIN {X 94.180,Y 101.239,Z 88.997,A 180.000,B 0.000,C 180.000} C_DIS
LIN {X 100.817,Y 101.239,Z 89.000,A 180.000,B 0.000,C 180.000} C_DIS
LIN {X 101.087,Y 101.239,Z 88.611,A 180.000,B 0.000,C 180.000} C_DIS
LIN {X 101.688,Y 101.239,Z 87.676,A 180.000,B 0.000,C 180.000} C_DIS
LIN {X 102.052,Y 101.239,Z 87.091,A 180.000,B 0.000,C 180.000} C_DIS
LIN {X 102.495,Y 101.239,Z 86.335,A 180.000,B 0.000,C 180.000} C_DIS
LIN {X 103.118,Y 101.239,Z 85.247,A 180.000,B 0.000,C 180.000} C_DIS
LIN {X 103.612,Y 101.239,Z 84.355,A 180.000,B 0.000,C 180.000} C_DIS
LIN {X 104.340,Y 101.239,Z 82.999,A 180.000,B 0.000,C 180.000} C_DIS
LIN {X 105.204,Y 101.239,Z 81.359,A 180.000,B 0.000,C 180.000} C_DIS
LIN {X 106.349,Y 101.239,Z 79.118,A 180.000,B 0.000,C 180.000} C_DIS
LIN {X 108.116,Y 101.239,Z 75.584,A 180.000,B 0.000,C 180.000} C_DIS
LIN {X 110.238,Y 101.239,Z 71.253,A 180.000,B 0.000,C 180.000} C_DIS
LIN {X 112.019,Y 101.239,Z 67.560,A 180.000,B 0.000,C 180.000} C_DIS
LIN {X 112.022,Y 101.239,Z 62.000,A 180.000,B 0.000,C 180.000} C_DIS
LIN {X 122.297,Y 101.239,Z 62.000,A 180.000,B 0.000,C 180.000} C_DIS
LIN {X 122.297,Y 101.239,Z 57.000,A 180.000,B 0.000,C 180.000} C_DIS
LIN {X 148.640,Y 101.239,Z 57.000,A 180.000,B 0.000,C 180.000} C_DIS
LIN {X 148.640,Y 101.239,Z 52.000,A 180.000,B 0.000,C 180.000} C_DIS
LIN {X 152.500,Y 101.239,Z 52.000,A 180.000,B 0.000,C 180.000} C_DIS
LIN {X 152.500,Y 101.239,Z 45.000,A 180.000,B 0.000,C 180.000} C_DIS
LIN {X 155.010,Y 101.239,Z 45.000,A 180.000,B 0.000,C 180.000} C_DIS
; Link Move Starts
LIN {X 155.120,Y 101.239,Z 45.026,A 180.000,B 0.000,C 180.000} C_DIS
LIN {X 155.230,Y 101.239,Z 45.051,A 180.000,B 0.000,C 180.000} C_DIS
LIN {X 155.771,Y 101.551,Z 45.051,A 180.000,B 0.000,C 180.000} C_DIS
LIN {X 155.771,Y 102.176,Z 45.051,A 180.000,B 0.000,C 180.000} C_DIS
LIN {X 155.230,Y 102.488,Z 45.051,A 180.000,B 0.000,C 180.000} C_DIS
LIN {X 155.120,Y 102.488,Z 45.026,A 180.000,B 0.000,C 180.000} C_DIS
LIN {X 155.010,Y 102.488,Z 45.000,A 180.000,B 0.000,C 180.000} C_DIS
; Cutting Move Starts
LIN {X 152.500,Y 102.488,Z 45.000,A 180.000,B 0.000,C 180.000} C_DIS
LIN {X 152.500,Y 102.488,Z 52.000,A 180.000,B 0.000,C 180.000} C_DIS
LIN {X 148.209,Y 102.488,Z 52.000,A 180.000,B 0.000,C 180.000} C_DIS
LIN {X 148.209,Y 102.488,Z 57.000,A 180.000,B 0.000,C 180.000} C_DIS
LIN {X 121.047,Y 102.488,Z 57.000,A 180.000,B 0.000,C 180.000} C_DIS
LIN {X 121.044,Y 102.488,Z 62.000,A 180.000,B 0.000,C 180.000} C_DIS
LIN {X 111.646,Y 102.488,Z 62.000,A 180.000,B 0.000,C 180.000} C_DIS
LIN {X 111.643,Y 102.488,Z 67.562,A 180.000,B 0.000,C 180.000} C_DIS
LIN {X 109.418,Y 102.488,Z 72.015,A 180.000,B 0.000,C 180.000} C_DIS
LIN {X 107.786,Y 102.488,Z 75.205,A 180.000,B 0.000,C 180.000} C_DIS
LIN {X 106.556,Y 102.488,Z 77.546,A 180.000,B 0.000,C 180.000} C_DIS
LIN {X 105.788,Y 102.488,Z 78.973,A 180.000,B 0.000,C 180.000} C_DIS
LIN {X 105.278,Y 102.488,Z 79.904,A 180.000,B 0.000,C 180.000} C_DIS
LIN {X 104.587,Y 102.488,Z 81.132,A 180.000,B 0.000,C 180.000} C_DIS
LIN {X 103.757,Y 102.488,Z 82.561,A 180.000,B 0.000,C 180.000} C_DIS
LIN {X 103.179,Y 102.488,Z 83.510,A 180.000,B 0.000,C 180.000} C_DIS
LIN {X 102.365,Y 102.488,Z 84.779,A 180.000,B 0.000,C 180.000} C_DIS
LIN {X 101.971,Y 102.488,Z 85.354,A 180.000,B 0.000,C 180.000} C_DIS
LIN {X 101.309,Y 102.488,Z 86.261,A 180.000,B 0.000,C 180.000} C_DIS
LIN {X 101.011,Y 102.488,Z 86.639,A 180.000,B 0.000,C 180.000} C_DIS
LIN {X 100.655,Y 102.488,Z 87.055,A 180.000,B 0.000,C 180.000} C_DIS
LIN {X 100.341,Y 102.488,Z 87.410,A 180.000,B 0.000,C 180.000} C_DIS
LIN {X 100.099,Y 102.488,Z 87.658,A 180.000,B 0.000,C 180.000} C_DIS
LIN {X 99.586,Y 102.488,Z 88.125,A 180.000,B 0.000,C 180.000} C_DIS
LIN {X 99.383,Y 102.488,Z 88.287,A 180.000,B 0.000,C 180.000} C_DIS
LIN {X 99.011,Y 102.488,Z 88.536,A 180.000,B 0.000,C 180.000} C_DIS
LIN {X 98.820,Y 102.488,Z 88.656,A 180.000,B 0.000,C 180.000} C_DIS
LIN {X 98.623,Y 102.488,Z 88.752,A 180.000,B 0.000,C 180.000} C_DIS
LIN {X 98.212,Y 102.488,Z 88.915,A 180.000,B 0.000,C 180.000} C_DIS
LIN {X 98.025,Y 102.488,Z 88.963,A 180.000,B 0.000,C 180.000} C_DIS
LIN {X 97.755,Y 102.488,Z 89.000,A 180.000,B 0.000,C 180.000} C_DIS
LIN {X 97.210,Y 102.488,Z 88.996,A 180.000,B 0.000,C 180.000} C_DIS
LIN {X 96.922,Y 102.488,Z 88.953,A 180.000,B 0.000,C 180.000} C_DIS
LIN {X 96.729,Y 102.488,Z 88.894,A 180.000,B 0.000,C 180.000} C_DIS
LIN {X 96.305,Y 102.488,Z 88.721,A 180.000,B 0.000,C 180.000} C_DIS
LIN {X 96.133,Y 102.488,Z 88.629,A 180.000,B 0.000,C 180.000} C_DIS
LIN {X 95.660,Y 102.488,Z 88.317,A 180.000,B 0.000,C 180.000} C_DIS
LIN {X 95.468,Y 102.488,Z 88.171,A 180.000,B 0.000,C 180.000} C_DIS
LIN {X 95.223,Y 102.488,Z 87.954,A 180.000,B 0.000,C 180.000} C_DIS
LIN {X 94.876,Y 102.488,Z 87.633,A 180.000,B 0.000,C 180.000} C_DIS
LIN {X 94.604,Y 102.488,Z 87.350,A 180.000,B 0.000,C 180.000} C_DIS
LIN {X 94.066,Y 102.488,Z 86.731,A 180.000,B 0.000,C 180.000} C_DIS
LIN {X 93.769,Y 102.488,Z 86.361,A 180.000,B 0.000,C 180.000} C_DIS
LIN {X 93.448,Y 102.488,Z 85.932,A 180.000,B 0.000,C 180.000} C_DIS
LIN {X 92.952,Y 102.488,Z 85.245,A 180.000,B 0.000,C 180.000} C_DIS
LIN {X 92.544,Y 102.488,Z 84.640,A 180.000,B 0.000,C 180.000} C_DIS
LIN {X 91.755,Y 102.488,Z 83.404,A 180.000,B 0.000,C 180.000} C_DIS
LIN {X 91.220,Y 102.488,Z 82.522,A 180.000,B 0.000,C 180.000} C_DIS
LIN {X 90.364,Y 102.488,Z 81.047,A 180.000,B 0.000,C 180.000} C_DIS
LIN {X 89.514,Y 102.488,Z 79.530,A 180.000,B 0.000,C 180.000} C_DIS
LIN {X 88.511,Y 102.488,Z 77.671,A 180.000,B 0.000,C 180.000} C_DIS
LIN {X 87.672,Y 102.488,Z 76.079,A 180.000,B 0.000,C 180.000} C_DIS
LIN {X 86.970,Y 102.488,Z 74.733,A 180.000,B 0.000,C 180.000} C_DIS
LIN {X 85.399,Y 102.488,Z 71.652,A 180.000,B 0.000,C 180.000} C_DIS
LIN {X 83.354,Y 102.488,Z 67.555,A 180.000,B 0.000,C 180.000} C_DIS
LIN {X 83.353,Y 102.488,Z 62.000,A 180.000,B 0.000,C 180.000} C_DIS
LIN {X 71.008,Y 102.488,Z 62.000,A 180.000,B 0.000,C 180.000} C_DIS
LIN {X 71.003,Y 102.488,Z 66.500,A 180.000,B 0.000,C 180.000} C_DIS
LIN {X 70.957,Y 102.488,Z 66.500,A 180.000,B 0.000,C 180.000} C_DIS
LIN {X 70.957,Y 102.488,Z 70.000,A 180.000,B 0.000,C 180.000} C_DIS
LIN {X 65.985,Y 102.488,Z 70.000,A 180.000,B 0.000,C 180.000} C_DIS
LIN {X 65.983,Y 102.488,Z 74.500,A 180.000,B 0.000,C 180.000} C_DIS
LIN {X 65.935,Y 102.488,Z 74.500,A 180.000,B 0.000,C 180.000} C_DIS
LIN {X 65.935,Y 102.488,Z 78.000,A 180.000,B 0.000,C 180.000} C_DIS
LIN {X 51.070,Y 102.488,Z 78.000,A 180.000,B 0.000,C 180.000} C_DIS
LIN {X 51.070,Y 102.488,Z 74.500,A 180.000,B 0.000,C 180.000} C_DIS
LIN {X 51.020,Y 102.488,Z 74.500,A 180.000,B 0.000,C 180.000} C_DIS
LIN {X 51.020,Y 102.488,Z 70.000,A 180.000,B 0.000,C 180.000} C_DIS
LIN {X 46.043,Y 102.488,Z 70.000,A 180.000,B 0.000,C 180.000} C_DIS
LIN {X 46.043,Y 102.488,Z 66.500,A 180.000,B 0.000,C 180.000} C_DIS
LIN {X 45.992,Y 102.488,Z 66.500,A 180.000,B 0.000,C 180.000} C_DIS
LIN {X 45.992,Y 102.488,Z 62.000,A 180.000,B 0.000,C 180.000} C_DIS
LIN {X 33.953,Y 102.488,Z 62.000,A 180.000,B 0.000,C 180.000} C_DIS
LIN {X 33.953,Y 102.488,Z 57.000,A 180.000,B 0.000,C 180.000} C_DIS
LIN {X 6.791,Y 102.488,Z 57.000,A 180.000,B 0.000,C 180.000} C_DIS
LIN {X 6.790,Y 102.488,Z 52.000,A 180.000,B 0.000,C 180.000} C_DIS
LIN {X 2.500,Y 102.488,Z 52.000,A 180.000,B 0.000,C 180.000} C_DIS
LIN {X 2.500,Y 102.488,Z 45.000,A 180.000,B 0.000,C 180.000} C_DIS
LIN {X -0.010,Y 102.488,Z 45.000,A 180.000,B 0.000,C 180.000} C_DIS
; Link Move Starts
LIN {X -0.120,Y 102.488,Z 45.026,A 180.000,B 0.000,C 180.000} C_DIS
LIN {X -0.230,Y 102.488,Z 45.051,A 180.000,B 0.000,C 180.000} C_DIS
LIN {X -0.771,Y 102.801,Z 45.051,A 180.000,B 0.000,C 180.000} C_DIS
LIN {X -0.771,Y 103.426,Z 45.051,A 180.000,B 0.000,C 180.000} C_DIS
LIN {X -0.230,Y 103.738,Z 45.051,A 180.000,B 0.000,C 180.000} C_DIS
LIN {X -0.120,Y 103.738,Z 45.026,A 180.000,B 0.000,C 180.000} C_DIS
LIN {X -0.010,Y 103.738,Z 45.000,A 180.000,B 0.000,C 180.000} C_DIS
; Cutting Move Starts
LIN {X 2.497,Y 103.738,Z 45.000,A 180.000,B 0.000,C 180.000} C_DIS
LIN {X 2.500,Y 103.738,Z 52.000,A 180.000,B 0.000,C 180.000} C_DIS
LIN {X 7.243,Y 103.738,Z 52.000,A 180.000,B 0.000,C 180.000} C_DIS
LIN {X 7.243,Y 103.738,Z 57.000,A 180.000,B 0.000,C 180.000} C_DIS
LIN {X 35.203,Y 103.738,Z 57.000,A 180.000,B 0.000,C 180.000} C_DIS
LIN {X 35.203,Y 103.738,Z 62.000,A 180.000,B 0.000,C 180.000} C_DIS
LIN {X 46.153,Y 103.738,Z 62.000,A 180.000,B 0.000,C 180.000} C_DIS
LIN {X 46.153,Y 103.738,Z 66.500,A 180.000,B 0.000,C 180.000} C_DIS
LIN {X 46.204,Y 103.738,Z 66.500,A 180.000,B 0.000,C 180.000} C_DIS
LIN {X 46.204,Y 103.738,Z 70.000,A 180.000,B 0.000,C 180.000} C_DIS
LIN {X 51.294,Y 103.738,Z 70.000,A 180.000,B 0.000,C 180.000} C_DIS
LIN {X 51.294,Y 103.738,Z 74.500,A 180.000,B 0.000,C 180.000} C_DIS
LIN {X 51.347,Y 103.738,Z 74.500,A 180.000,B 0.000,C 180.000} C_DIS
LIN {X 51.347,Y 103.738,Z 78.000,A 180.000,B 0.000,C 180.000} C_DIS
LIN {X 65.654,Y 103.738,Z 78.000,A 180.000,B 0.000,C 180.000} C_DIS
LIN {X 65.658,Y 103.738,Z 74.500,A 180.000,B 0.000,C 180.000} C_DIS
LIN {X 65.710,Y 103.738,Z 74.500,A 180.000,B 0.000,C 180.000} C_DIS
LIN {X 65.710,Y 103.738,Z 70.000,A 180.000,B 0.000,C 180.000} C_DIS
LIN {X 70.792,Y 103.738,Z 70.000,A 180.000,B 0.000,C 180.000} C_DIS
LIN {X 70.796,Y 103.738,Z 66.500,A 180.000,B 0.000,C 180.000} C_DIS
LIN {X 70.847,Y 103.738,Z 66.500,A 180.000,B 0.000,C 180.000} C_DIS
LIN {X 70.847,Y 103.738,Z 62.000,A 180.000,B 0.000,C 180.000} C_DIS
LIN {X 83.864,Y 103.738,Z 62.000,A 180.000,B 0.000,C 180.000} C_DIS
LIN {X 83.864,Y 103.738,Z 67.555,A 180.000,B 0.000,C 180.000} C_DIS
LIN {X 84.466,Y 103.738,Z 68.734,A 180.000,B 0.000,C 180.000} C_DIS
LIN {X 86.180,Y 103.738,Z 72.003,A 180.000,B 0.000,C 180.000} C_DIS
LIN {X 87.521,Y 103.738,Z 74.485,A 180.000,B 0.000,C 180.000} C_DIS
LIN {X 88.649,Y 103.738,Z 76.498,A 180.000,B 0.000,C 180.000} C_DIS
LIN {X 89.653,Y 103.738,Z 78.224,A 180.000,B 0.000,C 180.000} C_DIS
LIN {X 90.389,Y 103.738,Z 79.435,A 180.000,B 0.000,C 180.000} C_DIS
LIN {X 91.295,Y 103.738,Z 80.852,A 180.000,B 0.000,C 180.000} C_DIS
LIN {X 91.883,Y 103.738,Z 81.720,A 180.000,B 0.000,C 180.000} C_DIS
LIN {X 92.574,Y 103.738,Z 82.672,A 180.000,B 0.000,C 180.000} C_DIS
LIN {X 92.977,Y 103.738,Z 83.197,A 180.000,B 0.000,C 180.000} C_DIS
LIN {X 93.265,Y 103.738,Z 83.548,A 180.000,B 0.000,C 180.000} C_DIS
LIN {X 93.669,Y 103.738,Z 84.016,A 180.000,B 0.000,C 180.000} C_DIS
LIN {X 94.010,Y 103.738,Z 84.393,A 180.000,B 0.000,C 180.000} C_DIS
LIN {X 94.290,Y 103.738,Z 84.674,A 180.000,B 0.000,C 180.000} C_DIS
LIN {X 94.599,Y 103.738,Z 84.960,A 180.000,B 0.000,C 180.000} C_DIS
LIN {X 94.926,Y 103.738,Z 85.249,A 180.000,B 0.000,C 180.000} C_DIS
LIN {X 95.194,Y 103.738,Z 85.458,A 180.000,B 0.000,C 180.000} C_DIS
LIN {X 95.568,Y 103.738,Z 85.709,A 180.000,B 0.000,C 180.000} C_DIS
LIN {X 95.805,Y 103.738,Z 85.858,A 180.000,B 0.000,C 180.000} C_DIS
LIN {X 96.041,Y 103.738,Z 85.982,A 180.000,B 0.000,C 180.000} C_DIS
LIN {X 96.497,Y 103.738,Z 86.168,A 180.000,B 0.000,C 180.000} C_DIS
LIN {X 96.698,Y 103.738,Z 86.233,A 180.000,B 0.000,C 180.000} C_DIS
LIN {X 96.895,Y 103.738,Z 86.277,A 180.000,B 0.000,C 180.000} C_DIS
LIN {X 97.225,Y 103.738,Z 86.324,A 180.000,B 0.000,C 180.000} C_DIS
LIN {X 97.458,Y 103.738,Z 86.344,A 180.000,B 0.000,C 180.000} C_DIS
LIN {X 97.666,Y 103.738,Z 86.336,A 180.000,B 0.000,C 180.000} C_DIS
LIN {X 97.999,Y 103.738,Z 86.294,A 180.000,B 0.000,C 180.000} C_DIS
LIN {X 98.216,Y 103.738,Z 86.256,A 180.000,B 0.000,C 180.000} C_DIS
LIN {X 98.423,Y 103.738,Z 86.197,A 180.000,B 0.000,C 180.000} C_DIS
LIN {X 98.663,Y 103.738,Z 86.104,A 180.000,B 0.000,C 180.000} C_DIS
LIN {X 98.983,Y 103.738,Z 85.971,A 180.000,B 0.000,C 180.000} C_DIS
LIN {X 99.237,Y 103.738,Z 85.834,A 180.000,B 0.000,C 180.000} C_DIS
LIN {X 99.714,Y 103.738,Z 85.522,A 180.000,B 0.000,C 180.000} C_DIS
LIN {X 99.933,Y 103.738,Z 85.361,A 180.000,B 0.000,C 180.000} C_DIS
LIN {X 100.174,Y 103.738,Z 85.163,A 180.000,B 0.000,C 180.000} C_DIS
LIN {X 100.591,Y 103.738,Z 84.787,A 180.000,B 0.000,C 180.000} C_DIS
LIN {X 100.890,Y 103.738,Z 84.496,A 180.000,B 0.000,C 180.000} C_DIS
LIN {X 101.168,Y 103.738,Z 84.199,A 180.000,B 0.000,C 180.000} C_DIS
LIN {X 101.521,Y 103.738,Z 83.798,A 180.000,B 0.000,C 180.000} C_DIS
LIN {X 101.925,Y 103.738,Z 83.320,A 180.000,B 0.000,C 180.000} C_DIS
LIN {X 102.381,Y 103.738,Z 82.733,A 180.000,B 0.000,C 180.000} C_DIS
LIN {X 103.084,Y 103.738,Z 81.766,A 180.000,B 0.000,C 180.000} C_DIS
LIN {X 103.631,Y 103.738,Z 80.964,A 180.000,B 0.000,C 180.000} C_DIS
LIN {X 104.520,Y 103.738,Z 79.580,A 180.000,B 0.000,C 180.000} C_DIS
LIN {X 105.309,Y 103.738,Z 78.288,A 180.000,B 0.000,C 180.000} C_DIS
LIN {X 106.323,Y 103.738,Z 76.547,A 180.000,B 0.000,C 180.000} C_DIS
LIN {X 107.359,Y 103.738,Z 74.701,A 180.000,B 0.000,C 180.000} C_DIS
LIN {X 108.742,Y 103.738,Z 72.149,A 180.000,B 0.000,C 180.000} C_DIS
LIN {X 110.323,Y 103.738,Z 69.141,A 180.000,B 0.000,C 180.000} C_DIS
LIN {X 111.135,Y 103.738,Z 67.558,A 180.000,B 0.000,C 180.000} C_DIS
LIN {X 111.136,Y 103.738,Z 62.000,A 180.000,B 0.000,C 180.000} C_DIS
LIN {X 119.795,Y 103.738,Z 62.000,A 180.000,B 0.000,C 180.000} C_DIS
LIN {X 119.797,Y 103.738,Z 57.000,A 180.000,B 0.000,C 180.000} C_DIS
LIN {X 147.756,Y 103.738,Z 57.000,A 180.000,B 0.000,C 180.000} C_DIS
LIN {X 147.757,Y 103.738,Z 52.000,A 180.000,B 0.000,C 180.000} C_DIS
LIN {X 152.500,Y 103.738,Z 52.000,A 180.000,B 0.000,C 180.000} C_DIS
LIN {X 152.500,Y 103.738,Z 45.000,A 180.000,B 0.000,C 180.000} C_DIS
LIN {X 155.010,Y 103.738,Z 45.000,A 180.000,B 0.000,C 180.000} C_DIS
; Link Move Starts
LIN {X 155.120,Y 103.738,Z 45.026,A 180.000,B 0.000,C 180.000} C_DIS
LIN {X 155.230,Y 103.738,Z 45.051,A 180.000,B 0.000,C 180.000} C_DIS
LIN {X 155.771,Y 104.051,Z 45.051,A 180.000,B 0.000,C 180.000} C_DIS
LIN {X 155.771,Y 104.676,Z 45.051,A 180.000,B 0.000,C 180.000} C_DIS
LIN {X 155.230,Y 104.988,Z 45.051,A 180.000,B 0.000,C 180.000} C_DIS
LIN {X 155.120,Y 104.988,Z 45.026,A 180.000,B 0.000,C 180.000} C_DIS
LIN {X 155.010,Y 104.988,Z 45.000,A 180.000,B 0.000,C 180.000} C_DIS
; Cutting Move Starts
LIN {X 152.500,Y 104.988,Z 45.000,A 180.000,B 0.000,C 180.000} C_DIS
LIN {X 152.500,Y 104.988,Z 52.000,A 180.000,B 0.000,C 180.000} C_DIS
LIN {X 147.281,Y 104.988,Z 52.000,A 180.000,B 0.000,C 180.000} C_DIS
LIN {X 147.281,Y 104.988,Z 57.000,A 180.000,B 0.000,C 180.000} C_DIS
LIN {X 118.547,Y 104.988,Z 57.000,A 180.000,B 0.000,C 180.000} C_DIS
LIN {X 118.547,Y 104.988,Z 62.000,A 180.000,B 0.000,C 180.000} C_DIS
LIN {X 110.492,Y 104.988,Z 62.000,A 180.000,B 0.000,C 180.000} C_DIS
LIN {X 110.492,Y 104.988,Z 67.555,A 180.000,B 0.000,C 180.000} C_DIS
LIN {X 109.339,Y 104.988,Z 69.680,A 180.000,B 0.000,C 180.000} C_DIS
LIN {X 108.039,Y 104.988,Z 71.995,A 180.000,B 0.000,C 180.000} C_DIS
LIN {X 106.821,Y 104.988,Z 74.082,A 180.000,B 0.000,C 180.000} C_DIS
LIN {X 105.883,Y 104.988,Z 75.615,A 180.000,B 0.000,C 180.000} C_DIS
LIN {X 104.898,Y 104.988,Z 77.148,A 180.000,B 0.000,C 180.000} C_DIS
LIN {X 104.193,Y 104.988,Z 78.183,A 180.000,B 0.000,C 180.000} C_DIS
LIN {X 103.409,Y 104.988,Z 79.264,A 180.000,B 0.000,C 180.000} C_DIS
LIN {X 102.810,Y 104.988,Z 80.036,A 180.000,B 0.000,C 180.000} C_DIS
LIN {X 102.287,Y 104.988,Z 80.657,A 180.000,B 0.000,C 180.000} C_DIS
LIN {X 101.965,Y 104.988,Z 81.021,A 180.000,B 0.000,C 180.000} C_DIS
LIN {X 101.598,Y 104.988,Z 81.416,A 180.000,B 0.000,C 180.000} C_DIS
LIN {X 101.182,Y 104.988,Z 81.823,A 180.000,B 0.000,C 180.000} C_DIS
LIN {X 100.797,Y 104.988,Z 82.169,A 180.000,B 0.000,C 180.000} C_DIS
LIN {X 100.533,Y 104.988,Z 82.396,A 180.000,B 0.000,C 180.000} C_DIS
LIN {X 100.178,Y 104.988,Z 82.665,A 180.000,B 0.000,C 180.000} C_DIS
LIN {X 99.621,Y 104.988,Z 83.031,A 180.000,B 0.000,C 180.000} C_DIS
LIN {X 99.318,Y 104.988,Z 83.196,A 180.000,B 0.000,C 180.000} C_DIS
LIN {X 99.126,Y 104.988,Z 83.283,A 180.000,B 0.000,C 180.000} C_DIS
LIN {X 98.674,Y 104.988,Z 83.465,A 180.000,B 0.000,C 180.000} C_DIS
LIN {X 98.365,Y 104.988,Z 83.557,A 180.000,B 0.000,C 180.000} C_DIS
LIN {X 98.065,Y 104.988,Z 83.611,A 180.000,B 0.000,C 180.000} C_DIS
LIN {X 97.754,Y 104.988,Z 83.651,A 180.000,B 0.000,C 180.000} C_DIS
LIN {X 97.541,Y 104.988,Z 83.663,A 180.000,B 0.000,C 180.000} C_DIS
LIN {X 97.292,Y 104.988,Z 83.654,A 180.000,B 0.000,C 180.000} C_DIS
LIN {X 97.073,Y 104.988,Z 83.630,A 180.000,B 0.000,C 180.000} C_DIS
LIN {X 96.820,Y 104.988,Z 83.592,A 180.000,B 0.000,C 180.000} C_DIS
LIN {X 96.608,Y 104.988,Z 83.550,A 180.000,B 0.000,C 180.000} C_DIS
LIN {X 96.304,Y 104.988,Z 83.457,A 180.000,B 0.000,C 180.000} C_DIS
LIN {X 95.828,Y 104.988,Z 83.264,A 180.000,B 0.000,C 180.000} C_DIS
